LIN {X 0,Y 580.1,Z 304.268,A -85,B 0,C 180,E1 -1819.83,E2 -1819.83} C_VEL
LIN {X 0,Y 580.128,Z 300.119,A -85,B 0,C 180,E1 -1822.058,E2 -1822.058} C_VEL
LIN {X 0,Y 580.155,Z 294.555,A -85,B 0,C 180,E1 -1825.087,E2 -1825.087} C_VEL
LIN {X 0,Y 580.133,Z 290.01,A -85,B 0,C 180,E1 -1827.41,E2 -1827.41} C_VEL
LIN {X 0,Y 580.063,Z 285.03,A -85,B 0,C 180,E1 -1829.785,E2 -1829.785} C_VEL
LIN {X 0,Y 580.054,Z 279.379,A -85,B 0,C 180,E1 -1832.216,E2 -1832.216} C_VEL
LIN {X 0,Y 580.077,Z 277.233,A -85,B 0,C 180,E1 -1833.103,E2 -1833.103} C_VEL
LIN {X 0,Y 580.282,Z 277.204,A -85,B 0,C 180,E1 -1834.697,E2 -1834.697} C_VEL
LIN {X 0,Y 580.301,Z 277.201,A -85,B 0,C 180,E1 -1837.268,E2 -1837.268} C_VEL
LIN {X 0,Y 580.292,Z 277.205,A -85,B 0,C 180,E1 -1840.27,E2 -1840.27} C_VEL
LIN {X 0,Y 580.264,Z 277.206,A -85,B 0,C 180,E1 -1842.708,E2 -1842.708} C_VEL
LIN {X 0,Y 580.273,Z 277.208,A -85,B 0,C 180,E1 -1845.609,E2 -1845.609} C_VEL
LIN {X 0,Y 580.278,Z 277.204,A -85,B 0,C 180,E1 -1848.669,E2 -1848.669} C_VEL
LIN {X 0,Y 580.274,Z 277.208,A -85,B 0,C 180,E1 -1850.964,E2 -1850.964} C_VEL
LIN {X 0,Y 580.309,Z 277.247,A -85,B 0,C 180,E1 -1853.219,E2 -1853.219} C_VEL
LIN {X 0,Y 580.988,Z 281.668,A -85,B 0,C 180,E1 -1854.504,E2 -1854.504} C_VEL
LIN {X 0,Y 580.826,Z 290.876,A -85,B 0,C 180,E1 -1857.009,E2 -1857.009} C_VEL
LIN {X 0,Y 580.744,Z 300.085,A -85,B 0,C 180,E1 -1859.451,E2 -1859.451} C_VEL
LIN {X 0,Y 580.649,Z 311.291,A -85,B 0,C 180,E1 -1862.344,E2 -1862.344} C_VEL
LIN {X 0,Y 580.515,Z 321.571,A -85,B 0,C 180,E1 -1864.93,E2 -1864.93} C_VEL
LIN {X 0,Y 580.444,Z 332.314,A -85,B 0,C 180,E1 -1867.579,E2 -1867.579} C_VEL
LIN {X 0,Y 580.362,Z 343.058,A -85,B 0,C 180,E1 -1870.18,E2 -1870.18} C_VEL
LIN {X 0,Y 580.308,Z 355.336,A -85,B 0,C 180,E1 -1873.102,E2 -1873.102} C_VEL
LIN {X 0,Y 580.195,Z 367.614,A -85,B 0,C 180,E1 -1875.98,E2 -1875.98} C_VEL
LIN {X 0,Y 580.152,Z 374.712,A -85,B 0,C 180,E1 -1877.627,E2 -1877.627} C_VEL
LIN {X 0,Y 580.817,Z 380.085,A -85,B 0,C 180,E1 -1877.73,E2 -1877.73} C_VEL
LIN {X 0,Y 580.72,Z 393.734,A -85,B 0,C 180,E1 -1878.061,E2 -1878.061} C_VEL
LIN {X 0,Y 580.617,Z 406.32,A -85,B 0,C 180,E1 -1878.515,E2 -1878.515} C_VEL
LIN {X 0,Y 580.487,Z 418.208,A -85,B 0,C 180,E1 -1879.095,E2 -1879.095} C_VEL
LIN {X 0,Y 580.451,Z 429.476,A -85,B 0,C 180,E1 -1879.8,E2 -1879.8} C_VEL
LIN {X 0,Y 580.352,Z 439.646,A -85,B 0,C 180,E1 -1880.591,E2 -1880.591} C_VEL
LIN {X 0,Y 580.279,Z 448.787,A -85,B 0,C 180,E1 -1881.468,E2 -1881.468} C_VEL
LIN {X 0,Y 580.199,Z 457.691,A -85,B 0,C 180,E1 -1882.518,E2 -1882.518} C_VEL
LIN {X 0,Y 580.12,Z 464.465,A -85,B 0,C 180,E1 -1883.505,E2 -1883.505} C_VEL
LIN {X 0,Y 580.139,Z 469.68,A -85,B 0,C 180,E1 -1884.438,E2 -1884.438} C_VEL
LIN {X 0,Y 580.108,Z 474.371,A -85,B 0,C 180,E1 -1885.483,E2 -1885.483} C_VEL
LIN {X 0,Y 580.123,Z 477.956,A -85,B 0,C 180,E1 -1886.527,E2 -1886.527} C_VEL
LIN {X 0,Y 580.043,Z 479.809,A -85,B 0,C 180,E1 -1887.222,E2 -1887.222} C_VEL
LIN {X 0,Y 580.04,Z 481.201,A -85,B 0,C 180,E1 -1887.917,E2 -1887.917} C_VEL
LIN {X 0,Y 580.04,Z 482.784,A -85,B 0,C 180,E1 -1889.306,E2 -1889.306} C_VEL
LIN {X 0,Y 580.037,Z 483,A -85,B 0,C 180,E1 -1890,E2 -1890} C_VEL
LIN {X 0,Y 580.047,Z 482.185,A -85,B 0,C 180,E1 -1891.389,E2 -1891.389} C_VEL
LIN {X 0,Y 580.04,Z 481.202,A -85,B 0,C 180,E1 -1892.083,E2 -1892.083} C_VEL
LIN {X 0,Y 580.043,Z 479.809,A -85,B 0,C 180,E1 -1892.778,E2 -1892.778} C_VEL
LIN {X 0,Y 580.11,Z 476.896,A -85,B 0,C 180,E1 -1893.821,E2 -1893.821} C_VEL
LIN {X 0,Y 580.053,Z 472.949,A -85,B 0,C 180,E1 -1894.865,E2 -1894.865} C_VEL
LIN {X 0,Y 580.139,Z 466.877,A -85,B 0,C 180,E1 -1896.085,E2 -1896.085} C_VEL
LIN {X 0,Y 580.184,Z 460.236,A -85,B 0,C 180,E1 -1897.132,E2 -1897.132} C_VEL
LIN {X 0,Y 580.25,Z 451.989,A -85,B 0,C 180,E1 -1898.182,E2 -1898.182} C_VEL
LIN {X 0,Y 580.308,Z 443.537,A -85,B 0,C 180,E1 -1899.058,E2 -1899.058} C_VEL
LIN {X 0,Y 580.417,Z 433.093,A -85,B 0,C 180,E1 -1899.936,E2 -1899.936} C_VEL
LIN {X 0,Y 580.475,Z 422.758,A -85,B 0,C 180,E1 -1900.64,E2 -1900.64} C_VEL
LIN {X 0,Y 580.563,Z 411.592,A -85,B 0,C 180,E1 -1901.248,E2 -1901.248} C_VEL
LIN {X 0,Y 580.628,Z 399.765,A -85,B 0,C 180,E1 -1901.742,E2 -1901.742} C_VEL
LIN {X 0,Y 580.766,Z 386.349,A -85,B 0,C 180,E1 -1902.138,E2 -1902.138} C_VEL
LIN {X 0,Y 580.611,Z 377.609,A -85,B 0,C 180,E1 -1902.318,E2 -1902.318} C_VEL
LIN {X 0,Y 580.153,Z 374.712,A -85,B 0,C 180,E1 -1902.373,E2 -1902.373} C_VEL
LIN {X 0,Y 580.234,Z 363.009,A -85,B 0,C 180,E1 -1905.095,E2 -1905.095} C_VEL
LIN {X 0,Y 580.326,Z 350.731,A -85,B 0,C 180,E1 -1907.988,E2 -1907.988} C_VEL
LIN {X 0,Y 580.403,Z 338.679,A -85,B 0,C 180,E1 -1910.874,E2 -1910.874} C_VEL
LIN {X 0,Y 580.49,Z 327.71,A -85,B 0,C 180,E1 -1913.549,E2 -1913.549} C_VEL
LIN {X 0,Y 580.586,Z 315.432,A -85,B 0,C 180,E1 -1916.608,E2 -1916.608} C_VEL
LIN {X 0,Y 580.721,Z 304.562,A -85,B 0,C 180,E1 -1919.383,E2 -1919.383} C_VEL
LIN {X 0,Y 580.825,Z 293.946,A -85,B 0,C 180,E1 -1922.168,E2 -1922.168} C_VEL
LIN {X 0,Y 580.893,Z 284.737,A -85,B 0,C 180,E1 -1924.655,E2 -1924.655} C_VEL
LIN {X 0,Y 580.881,Z 280.446,A -85,B 0,C 180,E1 -1925.843,E2 -1925.843} C_VEL
LIN {X 0,Y 580.27,Z 277.208,A -85,B 0,C 180,E1 -1926.827,E2 -1926.827} C_VEL
LIN {X 0,Y 580.284,Z 277.205,A -85,B 0,C 180,E1 -1929.184,E2 -1929.184} C_VEL
LIN {X 0,Y 580.252,Z 277.203,A -85,B 0,C 180,E1 -1931.771,E2 -1931.771} C_VEL
LIN {X 0,Y 580.248,Z 277.211,A -85,B 0,C 180,E1 -1934.628,E2 -1934.628} C_VEL
LIN {X 0,Y 580.263,Z 277.201,A -85,B 0,C 180,E1 -1937.292,E2 -1937.292} C_VEL
LIN {X 0,Y 580.297,Z 277.203,A -85,B 0,C 180,E1 -1940.067,E2 -1940.067} C_VEL
LIN {X 0,Y 580.301,Z 277.196,A -85,B 0,C 180,E1 -1943.066,E2 -1943.066} C_VEL
LIN {X 0,Y 580.317,Z 277.2,A -85,B 0,C 180,E1 -1946.145,E2 -1946.145} C_VEL
LIN {X 0,Y 580.278,Z 277.199,A -85,B 0,C 180,E1 -1948.615,E2 -1948.615} C_VEL
LIN {X 0,Y 580.296,Z 277.199,A -85,B 0,C 180,E1 -1951.024,E2 -1951.024} C_VEL
LIN {X 0,Y 580.293,Z 277.204,A -85,B 0,C 180,E1 -1953.666,E2 -1953.666} C_VEL
LIN {X 0,Y 580.149,Z 277.224,A -85,B 0,C 180,E1 -1956.436,E2 -1956.436} C_VEL
LIN {X 0,Y 580.074,Z 277.231,A -85,B 0,C 180,E1 -1957.188,E2 -1957.188} C_VEL
LIN {X 0,Y 580.081,Z 279.813,A -85,B 0,C 180,E1 -1959.43,E2 -1959.43} C_VEL
LIN {X 0,Y 580.033,Z 283.328,A -85,B 0,C 180,E1 -1962.367,E2 -1962.367} C_VEL
LIN {X 0,Y 580.047,Z 285.965,A -85,B 0,C 180,E1 -1964.54,E2 -1964.54} C_VEL
LIN {X 0,Y 580.045,Z 288.602,A -85,B 0,C 180,E1 -1966.691,E2 -1966.691} C_VEL
LIN {X 0,Y 580.043,Z 290.118,A -85,B 0,C 180,E1 -1967.758,E2 -1967.758} C_VEL
LIN {X 0,Y 580.785,Z 296.369,A -85,B 0,C 180,E1 -1967.907,E2 -1967.907} C_VEL
LIN {X 0,Y 580.646,Z 309.747,A -85,B 0,C 180,E1 -1968.303,E2 -1968.303} C_VEL
LIN {X 0,Y 580.564,Z 320.592,A -85,B 0,C 180,E1 -1968.752,E2 -1968.752} C_VEL
LIN {X 0,Y 580.493,Z 331.974,A -85,B 0,C 180,E1 -1969.36,E2 -1969.36} C_VEL
LIN {X 0,Y 580.42,Z 342.507,A -85,B 0,C 180,E1 -1970.064,E2 -1970.064} C_VEL
LIN {X 0,Y 580.319,Z 353.054,A -85,B 0,C 180,E1 -1970.942,E2 -1970.942} C_VEL
LIN {X 0,Y 580.251,Z 361.571,A -85,B 0,C 180,E1 -1971.818,E2 -1971.818} C_VEL
LIN {X 0,Y 580.176,Z 368.64,A -85,B 0,C 180,E1 -1972.693,E2 -1972.693} C_VEL
LIN {X 0,Y 580.137,Z 375.587,A -85,B 0,C 180,E1 -1973.741,E2 -1973.741} C_VEL
LIN {X 0,Y 580.086,Z 381.161,A -85,B 0,C 180,E1 -1974.787,E2 -1974.787} C_VEL
LIN {X 0,Y 580.105,Z 385.527,A -85,B 0,C 180,E1 -1975.831,E2 -1975.831} C_VEL
LIN {X 0,Y 580.043,Z 389.694,A -85,B 0,C 180,E1 -1977.222,E2 -1977.222} C_VEL
LIN {X 0,Y 580.04,Z 391.135,A -85,B 0,C 180,E1 -1977.917,E2 -1977.917} C_VEL
LIN {X 0,Y 580.04,Z 392.757,A -85,B 0,C 180,E1 -1979.306,E2 -1979.306} C_VEL
LIN {X 0,Y 580.038,Z 392.996,A -85,B 0,C 180,E1 -1980,E2 -1980} C_VEL
LIN {X 0,Y 580.047,Z 392.229,A -85,B 0,C 180,E1 -1981.389,E2 -1981.389} C_VEL
LIN {X 0,Y 580.04,Z 391.278,A -85,B 0,C 180,E1 -1982.083,E2 -1982.083} C_VEL
LIN {X 0,Y 580.044,Z 389.883,A -85,B 0,C 180,E1 -1982.778,E2 -1982.778} C_VEL
LIN {X 0,Y 580.11,Z 387.011,A -85,B 0,C 180,E1 -1983.821,E2 -1983.821} C_VEL
LIN {X 0,Y 580.053,Z 383.122,A -85,B 0,C 180,E1 -1984.865,E2 -1984.865} C_VEL
LIN {X 0,Y 580.161,Z 378.1,A -85,B 0,C 180,E1 -1985.91,E2 -1985.91} C_VEL
LIN {X 0,Y 580.158,Z 371.776,A -85,B 0,C 180,E1 -1986.958,E2 -1986.958} C_VEL
LIN {X 0,Y 580.231,Z 363.836,A -85,B 0,C 180,E1 -1988.007,E2 -1988.007} C_VEL
LIN {X 0,Y 580.298,Z 355.752,A -85,B 0,C 180,E1 -1988.883,E2 -1988.883} C_VEL
LIN {X 0,Y 580.366,Z 345.921,A -85,B 0,C 180,E1 -1989.761,E2 -1989.761} C_VEL
LIN {X 0,Y 580.459,Z 334.898,A -85,B 0,C 180,E1 -1990.552,E2 -1990.552} C_VEL
LIN {X 0,Y 580.522,Z 324.063,A -85,B 0,C 180,E1 -1991.169,E2 -1991.169} C_VEL
LIN {X 0,Y 580.626,Z 312.523,A -85,B 0,C 180,E1 -1991.68,E2 -1991.68} C_VEL
LIN {X 0,Y 580.725,Z 300.605,A -85,B 0,C 180,E1 -1992.072,E2 -1992.072} C_VEL
LIN {X 0,Y 580.652,Z 293.717,A -85,B 0,C 180,E1 -1992.245,E2 -1992.245} C_VEL
LIN {X 0,Y 580.063,Z 289.894,A -85,B 0,C 180,E1 -1992.352,E2 -1992.352} C_VEL
LIN {X 0,Y 580.004,Z 286.954,A -85,B 0,C 180,E1 -1994.742,E2 -1994.742} C_VEL
LIN {X 0,Y 580.022,Z 283.684,A -85,B 0,C 180,E1 -1997.429,E2 -1997.429} C_VEL
LIN {X 0,Y 579.37,Z 283.014,A -85,B 0,C 180,E1 -1998.005,E2 -1998.005} C_VEL
LIN {X 0,Y 576.505,Z 282.007,A -85,B 0,C 180,E1 -1998.941,E2 -1998.941} C_VEL
LIN {X 0,Y 574.078,Z 281.214,A -85,B 0,C 180,E1 -1999.694,E2 -1999.694} C_VEL
LIN {X 0,Y 573.042,Z 280.574,A -85,B 0,C 180,E1 -2000.275,E2 -2000.275} C_VEL
LIN {X 0,Y 572.962,Z 280.347,A -85,B 0,C 180,E1 -2000.472,E2 -2000.472} C_VEL
LIN {X 0,Y 572.945,Z 278.247,A -85,B 0,C 180,E1 -2002.35,E2 -2002.35} C_VEL
LIN {X 0,Y 573.197,Z 278.087,A -85,B 0,C 180,E1 -2004.862,E2 -2004.862} C_VEL
LIN {X 0,Y 573.223,Z 278.081,A -85,B 0,C 180,E1 -2006.978,E2 -2006.978} C_VEL
LIN {X 0,Y 573.244,Z 278.074,A -85,B 0,C 180,E1 -2009.487,E2 -2009.487} C_VEL
LIN {X 0,Y 573.257,Z 278.078,A -85,B 0,C 180,E1 -2012.645,E2 -2012.645} C_VEL
LIN {X 0,Y 573.208,Z 278.078,A -85,B 0,C 180,E1 -2015.188,E2 -2015.188} C_VEL
LIN {X 0,Y 573.24,Z 278.079,A -85,B 0,C 180,E1 -2017.807,E2 -2017.807} C_VEL
LIN {X 0,Y 573.248,Z 278.077,A -85,B 0,C 180,E1 -2020.525,E2 -2020.525} C_VEL
LIN {X 0,Y 573.243,Z 278.076,A -85,B 0,C 180,E1 -2023.359,E2 -2023.359} C_VEL
LIN {X 0,Y 573.248,Z 278.076,A -85,B 0,C 180,E1 -2026.331,E2 -2026.331} C_VEL
LIN {X 0,Y 573.238,Z 278.076,A -85,B 0,C 180,E1 -2028.543,E2 -2028.543} C_VEL
LIN {X 0,Y 573.245,Z 278.078,A -85,B 0,C 180,E1 -2031.298,E2 -2031.298} C_VEL
LIN {X 0,Y 573.216,Z 278.082,A -85,B 0,C 180,E1 -2034.019,E2 -2034.019} C_VEL
LIN {X 0,Y 573.166,Z 278.255,A -85,B 0,C 180,E1 -2035.771,E2 -2035.771} C_VEL
LIN {X 0,Y 573.104,Z 282.816,A -85,B 0,C 180,E1 -2038.176,E2 -2038.176} C_VEL
LIN {X 0,Y 573.057,Z 287.256,A -85,B 0,C 180,E1 -2040.622,E2 -2040.622} C_VEL
LIN {X 0,Y 573.058,Z 291.597,A -85,B 0,C 180,E1 -2043.014,E2 -2043.014} C_VEL
LIN {X 0,Y 573.07,Z 295.867,A -85,B 0,C 180,E1 -2045.357,E2 -2045.357} C_VEL
LIN {X 0,Y 573.042,Z 299.961,A -85,B 0,C 180,E1 -2047.654,E2 -2047.654} C_VEL
LIN {X 0,Y 573.016,Z 304.101,A -85,B 0,C 180,E1 -2049.915,E2 -2049.915} C_VEL
LIN {X 0,Y 572.975,Z 308.248,A -85,B 0,C 180,E1 -2052.143,E2 -2052.143} C_VEL
LIN {X 0,Y 573,Z 313.778,A -85,B 0,C 180,E1 -2055.074,E2 -2055.074} C_VEL
LIN {X 0,Y 573.003,Z 318.682,A -85,B 0,C 180,E1 -2057.583,E2 -2057.583} C_VEL
LIN {X 0,Y 573.854,Z 325.38,A -85,B 0,C 180,E1 -2057.736,E2 -2057.736} C_VEL
LIN {X 0,Y 573.74,Z 337.077,A -85,B 0,C 180,E1 -2058.07,E2 -2058.07} C_VEL
LIN {X 0,Y 573.601,Z 347.726,A -85,B 0,C 180,E1 -2058.484,E2 -2058.484} C_VEL
LIN {X 0,Y 573.525,Z 359.272,A -85,B 0,C 180,E1 -2059.068,E2 -2059.068} C_VEL
LIN {X 0,Y 573.444,Z 371.328,A -85,B 0,C 180,E1 -2059.853,E2 -2059.853} C_VEL
LIN {X 0,Y 573.321,Z 381.079,A -85,B 0,C 180,E1 -2060.652,E2 -2060.652} C_VEL
LIN {X 0,Y 573.225,Z 389.959,A -85,B 0,C 180,E1 -2061.54,E2 -2061.54} C_VEL
LIN {X 0,Y 573.143,Z 397.316,A -85,B 0,C 180,E1 -2062.425,E2 -2062.425} C_VEL
LIN {X 0,Y 573.104,Z 403.818,A -85,B 0,C 180,E1 -2063.369,E2 -2063.369} C_VEL
LIN {X 0,Y 573.07,Z 409.452,A -85,B 0,C 180,E1 -2064.37,E2 -2064.37} C_VEL
LIN {X 0,Y 573.028,Z 414.2,A -85,B 0,C 180,E1 -2065.427,E2 -2065.427} C_VEL
LIN {X 0,Y 573.022,Z 417.834,A -85,B 0,C 180,E1 -2066.484,E2 -2066.484} C_VEL
LIN {X 0,Y 572.959,Z 419.672,A -85,B 0,C 180,E1 -2067.188,E2 -2067.188} C_VEL
LIN {X 0,Y 572.946,Z 422.142,A -85,B 0,C 180,E1 -2068.594,E2 -2068.594} C_VEL
LIN {X 0,Y 572.941,Z 422.751,A -85,B 0,C 180,E1 -2069.297,E2 -2069.297} C_VEL
LIN {X 0,Y 572.94,Z 422.811,A -85,B 0,C 180,E1 -2070.703,E2 -2070.703} C_VEL
LIN {X 0,Y 572.947,Z 422.242,A -85,B 0,C 180,E1 -2071.406,E2 -2071.406} C_VEL
LIN {X 0,Y 572.96,Z 419.898,A -85,B 0,C 180,E1 -2072.812,E2 -2072.812} C_VEL
LIN {X 0,Y 573.015,Z 417.024,A -85,B 0,C 180,E1 -2073.868,E2 -2073.868} C_VEL
LIN {X 0,Y 572.962,Z 413.114,A -85,B 0,C 180,E1 -2074.926,E2 -2074.926} C_VEL
LIN {X 0,Y 573.076,Z 408.064,A -85,B 0,C 180,E1 -2075.983,E2 -2075.983} C_VEL
LIN {X 0,Y 573.082,Z 401.729,A -85,B 0,C 180,E1 -2077.044,E2 -2077.044} C_VEL
LIN {X 0,Y 573.175,Z 393.872,A -85,B 0,C 180,E1 -2078.106,E2 -2078.106} C_VEL
LIN {X 0,Y 573.287,Z 383.962,A -85,B 0,C 180,E1 -2079.17,E2 -2079.17} C_VEL
LIN {X 0,Y 573.395,Z 374.773,A -85,B 0,C 180,E1 -2079.97,E2 -2079.97} C_VEL
LIN {X 0,Y 573.466,Z 364.905,A -85,B 0,C 180,E1 -2080.678,E2 -2080.678} C_VEL
LIN {X 0,Y 573.561,Z 352.657,A -85,B 0,C 180,E1 -2081.379,E2 -2081.379} C_VEL
LIN {X 0,Y 573.709,Z 339.914,A -85,B 0,C 180,E1 -2081.921,E2 -2081.921} C_VEL
LIN {X 0,Y 573.809,Z 328.042,A -85,B 0,C 180,E1 -2082.287,E2 -2082.287} C_VEL
LIN {X 0,Y 573.654,Z 322.803,A -85,B 0,C 180,E1 -2082.418,E2 -2082.418} C_VEL
LIN {X 0,Y 572.975,Z 318.53,A -85,B 0,C 180,E1 -2082.53,E2 -2082.53} C_VEL
LIN {X 0,Y 572.999,Z 313.949,A -85,B 0,C 180,E1 -2084.926,E2 -2084.926} C_VEL
LIN {X 0,Y 572.97,Z 308.416,A -85,B 0,C 180,E1 -2087.857,E2 -2087.857} C_VEL
LIN {X 0,Y 573.017,Z 304.267,A -85,B 0,C 180,E1 -2090.085,E2 -2090.085} C_VEL
LIN {X 0,Y 573.043,Z 300.122,A -85,B 0,C 180,E1 -2092.346,E2 -2092.346} C_VEL
LIN {X 0,Y 573.087,Z 294.611,A -85,B 0,C 180,E1 -2095.418,E2 -2095.418} C_VEL
LIN {X 0,Y 573.082,Z 289.95,A -85,B 0,C 180,E1 -2097.996,E2 -2097.996} C_VEL
LIN {X 0,Y 573.111,Z 284.493,A -85,B 0,C 180,E1 -2101,E2 -2101} C_VEL
LIN {X 0,Y 573.14,Z 279.854,A -85,B 0,C 180,E1 -2103.505,E2 -2103.505} C_VEL
LIN {X 0,Y 573.186,Z 278.091,A -85,B 0,C 180,E1 -2104.494,E2 -2104.494} C_VEL
LIN {X 0,Y 573.241,Z 278.084,A -85,B 0,C 180,E1 -2107.164,E2 -2107.164} C_VEL
LIN {X 0,Y 573.25,Z 278.081,A -85,B 0,C 180,E1 -2109.607,E2 -2109.607} C_VEL
LIN {X 0,Y 573.245,Z 278.081,A -85,B 0,C 180,E1 -2112.642,E2 -2112.642} C_VEL
LIN {X 0,Y 573.226,Z 278.082,A -85,B 0,C 180,E1 -2115.665,E2 -2115.665} C_VEL
LIN {X 0,Y 573.229,Z 278.082,A -85,B 0,C 180,E1 -2118.543,E2 -2118.543} C_VEL
LIN {X 0,Y 573.248,Z 278.081,A -85,B 0,C 180,E1 -2121.299,E2 -2121.299} C_VEL
LIN {X 0,Y 573.197,Z 278.089,A -85,B 0,C 180,E1 -2124.021,E2 -2124.021} C_VEL
LIN {X 0,Y 573.16,Z 278.132,A -85,B 0,C 180,E1 -2125.781,E2 -2125.781} C_VEL
LIN {X 0,Y 573.11,Z 284.453,A -85,B 0,C 180,E1 -2129.138,E2 -2129.138} C_VEL
LIN {X 0,Y 573.098,Z 290.134,A -85,B 0,C 180,E1 -2132.225,E2 -2132.225} C_VEL
LIN {X 0,Y 573.099,Z 295.565,A -85,B 0,C 180,E1 -2135.159,E2 -2135.159} C_VEL
LIN {X 0,Y 573.042,Z 299.964,A -85,B 0,C 180,E1 -2137.654,E2 -2137.654} C_VEL
LIN {X 0,Y 573.016,Z 304.101,A -85,B 0,C 180,E1 -2139.915,E2 -2139.915} C_VEL
LIN {X 0,Y 572.975,Z 308.248,A -85,B 0,C 180,E1 -2142.143,E2 -2142.143} C_VEL
LIN {X 0,Y 573,Z 313.777,A -85,B 0,C 180,E1 -2145.074,E2 -2145.074} C_VEL
LIN {X 0,Y 573.003,Z 318.741,A -85,B 0,C 180,E1 -2147.583,E2 -2147.583} C_VEL
LIN {X 0,Y 573.856,Z 325.326,A -85,B 0,C 180,E1 -2147.736,E2 -2147.736} C_VEL
LIN {X 0,Y 573.733,Z 337.39,A -85,B 0,C 180,E1 -2148.079,E2 -2148.079} C_VEL
LIN {X 0,Y 573.626,Z 349.625,A -85,B 0,C 180,E1 -2148.566,E2 -2148.566} C_VEL
LIN {X 0,Y 573.533,Z 360.687,A -85,B 0,C 180,E1 -2149.149,E2 -2149.149} C_VEL
LIN {X 0,Y 573.419,Z 371.271,A -85,B 0,C 180,E1 -2149.852,E2 -2149.852} C_VEL
LIN {X 0,Y 573.312,Z 379.078,A -85,B 0,C 180,E1 -2150.474,E2 -2150.474} C_VEL
LIN {X 0,Y 573.216,Z 388.327,A -85,B 0,C 180,E1 -2151.362,E2 -2151.362} C_VEL
LIN {X 0,Y 573.161,Z 395.962,A -85,B 0,C 180,E1 -2152.248,E2 -2152.248} C_VEL
LIN {X 0,Y 573.09,Z 403.915,A -85,B 0,C 180,E1 -2153.381,E2 -2153.381} C_VEL
LIN {X 0,Y 573.071,Z 409.462,A -85,B 0,C 180,E1 -2154.37,E2 -2154.37} C_VEL
LIN {X 0,Y 573.028,Z 414.203,A -85,B 0,C 180,E1 -2155.427,E2 -2155.427} C_VEL
LIN {X 0,Y 573.022,Z 417.833,A -85,B 0,C 180,E1 -2156.484,E2 -2156.484} C_VEL
LIN {X 0,Y 572.959,Z 419.688,A -85,B 0,C 180,E1 -2157.188,E2 -2157.188} C_VEL
LIN {X 0,Y 572.946,Z 422.135,A -85,B 0,C 180,E1 -2158.594,E2 -2158.594} C_VEL
LIN {X 0,Y 572.941,Z 422.758,A -85,B 0,C 180,E1 -2159.297,E2 -2159.297} C_VEL
LIN {X 0,Y 572.94,Z 422.805,A -85,B 0,C 180,E1 -2160.703,E2 -2160.703} C_VEL
LIN {X 0,Y 572.947,Z 422.244,A -85,B 0,C 180,E1 -2161.406,E2 -2161.406} C_VEL
LIN {X 0,Y 572.96,Z 419.895,A -85,B 0,C 180,E1 -2162.812,E2 -2162.812} C_VEL
LIN {X 0,Y 573.015,Z 417.023,A -85,B 0,C 180,E1 -2163.868,E2 -2163.868} C_VEL
LIN {X 0,Y 572.962,Z 413.115,A -85,B 0,C 180,E1 -2164.926,E2 -2164.926} C_VEL
LIN {X 0,Y 573.076,Z 408.065,A -85,B 0,C 180,E1 -2165.983,E2 -2165.983} C_VEL
LIN {X 0,Y 573.082,Z 401.724,A -85,B 0,C 180,E1 -2167.044,E2 -2167.044} C_VEL
LIN {X 0,Y 573.175,Z 393.869,A -85,B 0,C 180,E1 -2168.106,E2 -2168.106} C_VEL
LIN {X 0,Y 573.282,Z 383.983,A -85,B 0,C 180,E1 -2169.17,E2 -2169.17} C_VEL
LIN {X 0,Y 573.395,Z 374.778,A -85,B 0,C 180,E1 -2169.97,E2 -2169.97} C_VEL
LIN {X 0,Y 573.465,Z 364.906,A -85,B 0,C 180,E1 -2170.676,E2 -2170.676} C_VEL
LIN {X 0,Y 573.551,Z 354.024,A -85,B 0,C 180,E1 -2171.306,E2 -2171.306} C_VEL
LIN {X 0,Y 573.678,Z 341.003,A -85,B 0,C 180,E1 -2171.886,E2 -2171.886} C_VEL
LIN {X 0,Y 573.809,Z 328.053,A -85,B 0,C 180,E1 -2172.287,E2 -2172.287} C_VEL
LIN {X 0,Y 573.654,Z 322.819,A -85,B 0,C 180,E1 -2172.418,E2 -2172.418} C_VEL
LIN {X 0,Y 572.975,Z 318.53,A -85,B 0,C 180,E1 -2172.53,E2 -2172.53} C_VEL
LIN {X 0,Y 572.999,Z 313.949,A -85,B 0,C 180,E1 -2174.926,E2 -2174.926} C_VEL
LIN {X 0,Y 572.97,Z 308.416,A -85,B 0,C 180,E1 -2177.857,E2 -2177.857} C_VEL
LIN {X 0,Y 573.017,Z 304.267,A -85,B 0,C 180,E1 -2180.085,E2 -2180.085} C_VEL
LIN {X 0,Y 573.044,Z 300.135,A -85,B 0,C 180,E1 -2182.346,E2 -2182.346} C_VEL
LIN {X 0,Y 573.072,Z 295.562,A -85,B 0,C 180,E1 -2184.835,E2 -2184.835} C_VEL
LIN {X 0,Y 573.053,Z 291.375,A -85,B 0,C 180,E1 -2186.986,E2 -2186.986} C_VEL
LIN {X 0,Y 572.981,Z 286.225,A -85,B 0,C 180,E1 -2189.441,E2 -2189.441} C_VEL
LIN {X 0,Y 572.987,Z 280.726,A -85,B 0,C 180,E1 -2191.831,E2 -2191.831} C_VEL
LIN {X 0,Y 572.991,Z 278.115,A -85,B 0,C 180,E1 -2192.923,E2 -2192.923} C_VEL
LIN {X 0,Y 573.228,Z 278.083,A -85,B 0,C 180,E1 -2194.77,E2 -2194.77} C_VEL
LIN {X 0,Y 573.236,Z 278.084,A -85,B 0,C 180,E1 -2197.808,E2 -2197.808} C_VEL
LIN {X 0,Y 573.248,Z 278.082,A -85,B 0,C 180,E1 -2200.525,E2 -2200.525} C_VEL
LIN {X 0,Y 573.244,Z 278.08,A -85,B 0,C 180,E1 -2203.669,E2 -2203.669} C_VEL
LIN {X 0,Y 573.235,Z 278.081,A -85,B 0,C 180,E1 -2206.64,E2 -2206.64} C_VEL
LIN {X 0,Y 573.247,Z 278.083,A -85,B 0,C 180,E1 -2209.475,E2 -2209.475} C_VEL
LIN {X 0,Y 573.236,Z 278.084,A -85,B 0,C 180,E1 -2212.192,E2 -2212.192} C_VEL
LIN {X 0,Y 573.263,Z 278.145,A -85,B 0,C 180,E1 -2212.957,E2 -2212.957} C_VEL
LIN {X 0,Y 574.098,Z 283.202,A -85,B 0,C 180,E1 -2214.445,E2 -2214.445} C_VEL
LIN {X 0,Y 573.899,Z 292.411,A -85,B 0,C 180,E1 -2216.979,E2 -2216.979} C_VEL
LIN {X 0,Y 573.794,Z 301.619,A -85,B 0,C 180,E1 -2219.449,E2 -2219.449} C_VEL
LIN {X 0,Y 573.677,Z 312.363,A -85,B 0,C 180,E1 -2222.255,E2 -2222.255} C_VEL
LIN {X 0,Y 573.517,Z 323.417,A -85,B 0,C 180,E1 -2225.069,E2 -2225.069} C_VEL
LIN {X 0,Y 573.42,Z 333.849,A -85,B 0,C 180,E1 -2227.67,E2 -2227.67} C_VEL
LIN {X 0,Y 573.329,Z 346.127,A -85,B 0,C 180,E1 -2230.672,E2 -2230.672} C_VEL
LIN {X 0,Y 573.257,Z 357.095,A -85,B 0,C 180,E1 -2233.309,E2 -2233.309} C_VEL
LIN {X 0,Y 573.153,Z 369.148,A -85,B 0,C 180,E1 -2236.166,E2 -2236.166} C_VEL
LIN {X 0,Y 573.108,Z 374.712,A -85,B 0,C 180,E1 -2237.473,E2 -2237.473} C_VEL
LIN {X 0,Y 573.891,Z 381.227,A -85,B 0,C 180,E1 -2237.603,E2 -2237.603} C_VEL
LIN {X 0,Y 573.775,Z 394.495,A -85,B 0,C 180,E1 -2237.937,E2 -2237.937} C_VEL
LIN {X 0,Y 573.644,Z 407.393,A -85,B 0,C 180,E1 -2238.421,E2 -2238.421} C_VEL
LIN {X 0,Y 573.52,Z 419.994,A -85,B 0,C 180,E1 -2239.063,E2 -2239.063} C_VEL
LIN {X 0,Y 573.45,Z 430.746,A -85,B 0,C 180,E1 -2239.764,E2 -2239.764} C_VEL
LIN {X 0,Y 573.308,Z 439.646,A -85,B 0,C 180,E1 -2240.474,E2 -2240.474} C_VEL
LIN {X 0,Y 573.215,Z 448.787,A -85,B 0,C 180,E1 -2241.362,E2 -2241.362} C_VEL
LIN {X 0,Y 573.142,Z 457.69,A -85,B 0,C 180,E1 -2242.425,E2 -2242.425} C_VEL
LIN {X 0,Y 573.051,Z 464.405,A -85,B 0,C 180,E1 -2243.415,E2 -2243.415} C_VEL
LIN {X 0,Y 573.07,Z 469.68,A -85,B 0,C 180,E1 -2244.37,E2 -2244.37} C_VEL
LIN {X 0,Y 573.028,Z 474.371,A -85,B 0,C 180,E1 -2245.427,E2 -2245.427} C_VEL
LIN {X 0,Y 573.022,Z 477.956,A -85,B 0,C 180,E1 -2246.484,E2 -2246.484} C_VEL
LIN {X 0,Y 572.959,Z 479.809,A -85,B 0,C 180,E1 -2247.188,E2 -2247.188} C_VEL
LIN {X 0,Y 572.94,Z 481.201,A -85,B 0,C 180,E1 -2247.891,E2 -2247.891} C_VEL
LIN {X 0,Y 572.941,Z 482.784,A -85,B 0,C 180,E1 -2249.297,E2 -2249.297} C_VEL
LIN {X 0,Y 572.938,Z 483,A -85,B 0,C 180,E1 -2250,E2 -2250} C_VEL
LIN {X 0,Y 572.946,Z 482.185,A -85,B 0,C 180,E1 -2251.406,E2 -2251.406} C_VEL
LIN {X 0,Y 572.94,Z 481.201,A -85,B 0,C 180,E1 -2252.109,E2 -2252.109} C_VEL
LIN {X 0,Y 572.959,Z 479.81,A -85,B 0,C 180,E1 -2252.812,E2 -2252.812} C_VEL
LIN {X 0,Y 573.015,Z 476.896,A -85,B 0,C 180,E1 -2253.868,E2 -2253.868} C_VEL
LIN {X 0,Y 572.963,Z 472.949,A -85,B 0,C 180,E1 -2254.926,E2 -2254.926} C_VEL
LIN {X 0,Y 573.065,Z 466.877,A -85,B 0,C 180,E1 -2256.16,E2 -2256.16} C_VEL
LIN {X 0,Y 573.119,Z 460.236,A -85,B 0,C 180,E1 -2257.221,E2 -2257.221} C_VEL
LIN {X 0,Y 573.201,Z 451.989,A -85,B 0,C 180,E1 -2258.283,E2 -2258.283} C_VEL
LIN {X 0,Y 573.287,Z 443.537,A -85,B 0,C 180,E1 -2259.17,E2 -2259.17} C_VEL
LIN {X 0,Y 573.425,Z 433.093,A -85,B 0,C 180,E1 -2260.058,E2 -2260.058} C_VEL
LIN {X 0,Y 573.511,Z 421.536,A -85,B 0,C 180,E1 -2260.847,E2 -2260.847} C_VEL
LIN {X 0,Y 573.611,Z 409.878,A -85,B 0,C 180,E1 -2261.466,E2 -2261.466} C_VEL
LIN {X 0,Y 573.75,Z 397.174,A -85,B 0,C 180,E1 -2261.974,E2 -2261.974} C_VEL
LIN {X 0,Y 573.846,Z 384.519,A -85,B 0,C 180,E1 -2262.331,E2 -2262.331} C_VEL
LIN {X 0,Y 573.661,Z 378.329,A -85,B 0,C 180,E1 -2262.459,E2 -2262.459} C_VEL
LIN {X 0,Y 573.108,Z 374.712,A -85,B 0,C 180,E1 -2262.527,E2 -2262.527} C_VEL
LIN {X 0,Y 573.191,Z 363.009,A -85,B 0,C 180,E1 -2265.285,E2 -2265.285} C_VEL
LIN {X 0,Y 573.286,Z 352.266,A -85,B 0,C 180,E1 -2267.847,E2 -2267.847} C_VEL
LIN {X 0,Y 573.367,Z 339.988,A -85,B 0,C 180,E1 -2270.822,E2 -2270.822} C_VEL
LIN {X 0,Y 573.502,Z 327.71,A -85,B 0,C 180,E1 -2273.854,E2 -2273.854} C_VEL
LIN {X 0,Y 573.598,Z 316.972,A -85,B 0,C 180,E1 -2276.564,E2 -2276.564} C_VEL
LIN {X 0,Y 573.746,Z 306.224,A -85,B 0,C 180,E1 -2279.339,E2 -2279.339} C_VEL
LIN {X 0,Y 573.902,Z 294.954,A -85,B 0,C 180,E1 -2282.331,E2 -2282.331} C_VEL
LIN {X 0,Y 574.02,Z 285.623,A -85,B 0,C 180,E1 -2284.884,E2 -2284.884} C_VEL
LIN {X 0,Y 573.857,Z 281.439,A -85,B 0,C 180,E1 -2286.07,E2 -2286.07} C_VEL
LIN {X 0,Y 573.259,Z 278.082,A -85,B 0,C 180,E1 -2287.103,E2 -2287.103} C_VEL
LIN {X 0,Y 573.231,Z 278.079,A -85,B 0,C 180,E1 -2289.609,E2 -2289.609} C_VEL
LIN {X 0,Y 573.221,Z 278.086,A -85,B 0,C 180,E1 -2292.639,E2 -2292.639} C_VEL
LIN {X 0,Y 573.225,Z 278.078,A -85,B 0,C 180,E1 -2295.665,E2 -2295.665} C_VEL
LIN {X 0,Y 573.227,Z 278.084,A -85,B 0,C 180,E1 -2298.543,E2 -2298.543} C_VEL
LIN {X 0,Y 573.248,Z 278.075,A -85,B 0,C 180,E1 -2301.299,E2 -2301.299} C_VEL
LIN {X 0,Y 573.215,Z 278.087,A -85,B 0,C 180,E1 -2304.019,E2 -2304.019} C_VEL
LIN {X 0,Y 573.273,Z 278.073,A -85,B 0,C 180,E1 -2306.518,E2 -2306.518} C_VEL
LIN {X 0,Y 573.231,Z 278.079,A -85,B 0,C 180,E1 -2309.118,E2 -2309.118} C_VEL
LIN {X 0,Y 573.242,Z 278.083,A -85,B 0,C 180,E1 -2311.436,E2 -2311.436} C_VEL
LIN {X 0,Y 573.265,Z 278.078,A -85,B 0,C 180,E1 -2313.81,E2 -2313.81} C_VEL
LIN {X 0,Y 573.129,Z 278.097,A -85,B 0,C 180,E1 -2316.13,E2 -2316.13} C_VEL
LIN {X 0,Y 572.969,Z 278.362,A -85,B 0,C 180,E1 -2317.651,E2 -2317.651} C_VEL
LIN {X 0,Y 572.979,Z 279.813,A -85,B 0,C 180,E1 -2319.163,E2 -2319.163} C_VEL
LIN {X 0,Y 572.955,Z 282.45,A -85,B 0,C 180,E1 -2321.402,E2 -2321.402} C_VEL
LIN {X 0,Y 572.94,Z 285.087,A -85,B 0,C 180,E1 -2323.613,E2 -2323.613} C_VEL
LIN {X 0,Y 572.975,Z 288.603,A -85,B 0,C 180,E1 -2326.523,E2 -2326.523} C_VEL
LIN {X 0,Y 572.987,Z 289.894,A -85,B 0,C 180,E1 -2327.583,E2 -2327.583} C_VEL
LIN {X 0,Y 573.866,Z 296.399,A -85,B 0,C 180,E1 -2327.759,E2 -2327.759} C_VEL
LIN {X 0,Y 573.696,Z 309.748,A -85,B 0,C 180,E1 -2328.159,E2 -2328.159} C_VEL
LIN {X 0,Y 573.582,Z 320.583,A -85,B 0,C 180,E1 -2328.614,E2 -2328.614} C_VEL
LIN {X 0,Y 573.511,Z 330.701,A -85,B 0,C 180,E1 -2329.153,E2 -2329.153} C_VEL
LIN {X 0,Y 573.468,Z 340.043,A -85,B 0,C 180,E1 -2329.764,E2 -2329.764} C_VEL
LIN {X 0,Y 573.309,Z 349.056,A -85,B 0,C 180,E1 -2330.474,E2 -2330.474} C_VEL
LIN {X 0,Y 573.237,Z 358.373,A -85,B 0,C 180,E1 -2331.362,E2 -2331.362} C_VEL
LIN {X 0,Y 573.143,Z 367.361,A -85,B 0,C 180,E1 -2332.425,E2 -2332.425} C_VEL
LIN {X 0,Y 573.09,Z 373.912,A -85,B 0,C 180,E1 -2333.382,E2 -2333.382} C_VEL
LIN {X 0,Y 573.071,Z 379.438,A -85,B 0,C 180,E1 -2334.37,E2 -2334.37} C_VEL
LIN {X 0,Y 573.028,Z 384.165,A -85,B 0,C 180,E1 -2335.428,E2 -2335.428} C_VEL
LIN {X 0,Y 573.022,Z 387.792,A -85,B 0,C 180,E1 -2336.484,E2 -2336.484} C_VEL
LIN {X 0,Y 572.959,Z 389.689,A -85,B 0,C 180,E1 -2337.188,E2 -2337.188} C_VEL
LIN {X 0,Y 572.94,Z 391.136,A -85,B 0,C 180,E1 -2337.891,E2 -2337.891} C_VEL
LIN {X 0,Y 572.941,Z 392.755,A -85,B 0,C 180,E1 -2339.297,E2 -2339.297} C_VEL
LIN {X 0,Y 572.939,Z 392.996,A -85,B 0,C 180,E1 -2340,E2 -2340} C_VEL
LIN {X 0,Y 572.947,Z 392.227,A -85,B 0,C 180,E1 -2341.406,E2 -2341.406} C_VEL
LIN {X 0,Y 572.94,Z 391.279,A -85,B 0,C 180,E1 -2342.109,E2 -2342.109} C_VEL
LIN {X 0,Y 572.959,Z 389.874,A -85,B 0,C 180,E1 -2342.812,E2 -2342.812} C_VEL
LIN {X 0,Y 573.015,Z 387.004,A -85,B 0,C 180,E1 -2343.868,E2 -2343.868} C_VEL
LIN {X 0,Y 572.962,Z 383.117,A -85,B 0,C 180,E1 -2344.926,E2 -2344.926} C_VEL
LIN {X 0,Y 573.072,Z 378.097,A -85,B 0,C 180,E1 -2345.984,E2 -2345.984} C_VEL
LIN {X 0,Y 573.113,Z 370.536,A -85,B 0,C 180,E1 -2347.221,E2 -2347.221} C_VEL
LIN {X 0,Y 573.169,Z 363.826,A -85,B 0,C 180,E1 -2348.106,E2 -2348.106} C_VEL
LIN {X 0,Y 573.251,Z 355.737,A -85,B 0,C 180,E1 -2348.993,E2 -2348.993} C_VEL
LIN {X 0,Y 573.329,Z 346.965,A -85,B 0,C 180,E1 -2349.793,E2 -2349.793} C_VEL
LIN {X 0,Y 573.462,Z 336.257,A -85,B 0,C 180,E1 -2350.593,E2 -2350.593} C_VEL
LIN {X 0,Y 573.551,Z 324.052,A -85,B 0,C 180,E1 -2351.306,E2 -2351.306} C_VEL
LIN {X 0,Y 573.667,Z 312.485,A -85,B 0,C 180,E1 -2351.824,E2 -2351.824} C_VEL
LIN {X 0,Y 573.77,Z 301.328,A -85,B 0,C 180,E1 -2352.198,E2 -2352.198} C_VEL
LIN {X 0,Y 573.659,Z 294.448,A -85,B 0,C 180,E1 -2352.38,E2 -2352.38} C_VEL
LIN {X 0,Y 572.945,Z 289.893,A -85,B 0,C 180,E1 -2352.508,E2 -2352.508} C_VEL
LIN {X 0,Y 572.93,Z 286.953,A -85,B 0,C 180,E1 -2354.928,E2 -2354.928} C_VEL
LIN {X 0,Y 572.934,Z 283.436,A -85,B 0,C 180,E1 -2357.859,E2 -2357.859} C_VEL
LIN {X 0,Y 572.962,Z 280.347,A -85,B 0,C 180,E1 -2360.472,E2 -2360.472} C_VEL
LIN {X 0,Y 572.304,Z 279.767,A -85,B 0,C 180,E1 -2361.055,E2 -2361.055} C_VEL
LIN {X 0,Y 569.459,Z 279.212,A -85,B 0,C 180,E1 -2362.006,E2 -2362.006} C_VEL
LIN {X 0,Y 567.072,Z 279.031,A -85,B 0,C 180,E1 -2362.772,E2 -2362.772} C_VEL
LIN {X 0,Y 566.076,Z 278.986,A -85,B 0,C 180,E1 -2363.364,E2 -2363.364} C_VEL
LIN {X 0,Y 566.011,Z 278.981,A -85,B 0,C 180,E1 -2363.564,E2 -2363.564} C_VEL
LIN {X 0,Y 566.198,Z 278.951,A -85,B 0,C 180,E1 -2365.75,E2 -2365.75} C_VEL
LIN {X 0,Y 566.207,Z 278.954,A -85,B 0,C 180,E1 -2368.202,E2 -2368.202} C_VEL
LIN {X 0,Y 566.191,Z 278.953,A -85,B 0,C 180,E1 -2371.076,E2 -2371.076} C_VEL
LIN {X 0,Y 566.215,Z 278.951,A -85,B 0,C 180,E1 -2373.734,E2 -2373.734} C_VEL
LIN {X 0,Y 566.203,Z 278.956,A -85,B 0,C 180,E1 -2376.57,E2 -2376.57} C_VEL
LIN {X 0,Y 566.219,Z 278.952,A -85,B 0,C 180,E1 -2379.686,E2 -2379.686} C_VEL
LIN {X 0,Y 566.213,Z 278.959,A -85,B 0,C 180,E1 -2382.088,E2 -2382.088} C_VEL
LIN {X 0,Y 566.177,Z 278.955,A -85,B 0,C 180,E1 -2385.036,E2 -2385.036} C_VEL
LIN {X 0,Y 566.213,Z 278.958,A -85,B 0,C 180,E1 -2387.912,E2 -2387.912} C_VEL
LIN {X 0,Y 566.218,Z 278.95,A -85,B 0,C 180,E1 -2390.726,E2 -2390.726} C_VEL
LIN {X 0,Y 566.187,Z 278.96,A -85,B 0,C 180,E1 -2393.788,E2 -2393.788} C_VEL
LIN {X 0,Y 566.103,Z 279.08,A -85,B 0,C 180,E1 -2395.822,E2 -2395.822} C_VEL
LIN {X 0,Y 566.033,Z 284.284,A -85,B 0,C 180,E1 -2398.568,E2 -2398.568} C_VEL
LIN {X 0,Y 565.978,Z 288.692,A -85,B 0,C 180,E1 -2401.035,E2 -2401.035} C_VEL
LIN {X 0,Y 566.019,Z 293.024,A -85,B 0,C 180,E1 -2403.449,E2 -2403.449} C_VEL
LIN {X 0,Y 565.968,Z 297.287,A -85,B 0,C 180,E1 -2405.809,E2 -2405.809} C_VEL
LIN {X 0,Y 565.968,Z 302.336,A -85,B 0,C 180,E1 -2408.643,E2 -2408.643} C_VEL
LIN {X 0,Y 565.955,Z 306.867,A -85,B 0,C 180,E1 -2411.164,E2 -2411.164} C_VEL
LIN {X 0,Y 565.883,Z 312.396,A -85,B 0,C 180,E1 -2414.143,E2 -2414.143} C_VEL
LIN {X 0,Y 565.892,Z 316.544,A -85,B 0,C 180,E1 -2416.351,E2 -2416.351} C_VEL
LIN {X 0,Y 565.91,Z 318.663,A -85,B 0,C 180,E1 -2417.425,E2 -2417.425} C_VEL
LIN {X 0,Y 566.911,Z 325.394,A -85,B 0,C 180,E1 -2417.584,E2 -2417.584} C_VEL
LIN {X 0,Y 566.782,Z 337.074,A -85,B 0,C 180,E1 -2417.922,E2 -2417.922} C_VEL
LIN {X 0,Y 566.657,Z 347.721,A -85,B 0,C 180,E1 -2418.341,E2 -2418.341} C_VEL
LIN {X 0,Y 566.536,Z 358.159,A -85,B 0,C 180,E1 -2418.869,E2 -2418.869} C_VEL
LIN {X 0,Y 566.442,Z 368.851,A -85,B 0,C 180,E1 -2419.545,E2 -2419.545} C_VEL
LIN {X 0,Y 566.301,Z 379.134,A -85,B 0,C 180,E1 -2420.355,E2 -2420.355} C_VEL
LIN {X 0,Y 566.167,Z 388.335,A -85,B 0,C 180,E1 -2421.253,E2 -2421.253} C_VEL
LIN {X 0,Y 566.095,Z 395.943,A -85,B 0,C 180,E1 -2422.151,E2 -2422.151} C_VEL
LIN {X 0,Y 566.021,Z 402.805,A -85,B 0,C 180,E1 -2423.127,E2 -2423.127} C_VEL
LIN {X 0,Y 566,Z 409.455,A -85,B 0,C 180,E1 -2424.299,E2 -2424.299} C_VEL
LIN {X 0,Y 565.932,Z 414.204,A -85,B 0,C 180,E1 -2425.37,E2 -2425.37} C_VEL
LIN {X 0,Y 565.927,Z 417.838,A -85,B 0,C 180,E1 -2426.44,E2 -2426.44} C_VEL
LIN {X 0,Y 565.877,Z 419.669,A -85,B 0,C 180,E1 -2427.152,E2 -2427.152} C_VEL
LIN {X 0,Y 565.845,Z 422.144,A -85,B 0,C 180,E1 -2428.577,E2 -2428.577} C_VEL
LIN {X 0,Y 565.841,Z 422.751,A -85,B 0,C 180,E1 -2429.288,E2 -2429.288} C_VEL
LIN {X 0,Y 565.841,Z 422.81,A -85,B 0,C 180,E1 -2430.712,E2 -2430.712} C_VEL
LIN {X 0,Y 565.846,Z 422.243,A -85,B 0,C 180,E1 -2431.423,E2 -2431.423} C_VEL
LIN {X 0,Y 565.878,Z 419.892,A -85,B 0,C 180,E1 -2432.848,E2 -2432.848} C_VEL
LIN {X 0,Y 565.926,Z 417.015,A -85,B 0,C 180,E1 -2433.916,E2 -2433.916} C_VEL
LIN {X 0,Y 565.878,Z 413.103,A -85,B 0,C 180,E1 -2434.987,E2 -2434.987} C_VEL
LIN {X 0,Y 565.991,Z 408.052,A -85,B 0,C 180,E1 -2436.059,E2 -2436.059} C_VEL
LIN {X 0,Y 566.032,Z 401.717,A -85,B 0,C 180,E1 -2437.132,E2 -2437.132} C_VEL
LIN {X 0,Y 566.128,Z 393.87,A -85,B 0,C 180,E1 -2438.208,E2 -2438.208} C_VEL
LIN {X 0,Y 566.249,Z 383.945,A -85,B 0,C 180,E1 -2439.285,E2 -2439.285} C_VEL
LIN {X 0,Y 566.401,Z 374.754,A -85,B 0,C 180,E1 -2440.094,E2 -2440.094} C_VEL
LIN {X 0,Y 566.464,Z 364.976,A -85,B 0,C 180,E1 -2440.805,E2 -2440.805} C_VEL
LIN {X 0,Y 566.574,Z 354.064,A -85,B 0,C 180,E1 -2441.448,E2 -2441.448} C_VEL
LIN {X 0,Y 566.748,Z 341.293,A -85,B 0,C 180,E1 -2442.02,E2 -2442.02} C_VEL
LIN {X 0,Y 566.87,Z 328.862,A -85,B 0,C 180,E1 -2442.417,E2 -2442.417} C_VEL
LIN {X 0,Y 566.709,Z 323.446,A -85,B 0,C 180,E1 -2442.558,E2 -2442.558} C_VEL
LIN {X 0,Y 565.894,Z 318.596,A -85,B 0,C 180,E1 -2442.667,E2 -2442.667} C_VEL
LIN {X 0,Y 565.914,Z 313.948,A -85,B 0,C 180,E1 -2445.117,E2 -2445.117} C_VEL
LIN {X 0,Y 565.898,Z 308.415,A -85,B 0,C 180,E1 -2448.088,E2 -2448.088} C_VEL
LIN {X 0,Y 565.933,Z 304.272,A -85,B 0,C 180,E1 -2450.348,E2 -2450.348} C_VEL
LIN {X 0,Y 566.005,Z 299.121,A -85,B 0,C 180,E1 -2453.241,E2 -2453.241} C_VEL
LIN {X 0,Y 566.013,Z 294.629,A -85,B 0,C 180,E1 -2455.759,E2 -2455.759} C_VEL
LIN {X 0,Y 566.002,Z 290.297,A -85,B 0,C 180,E1 -2458.163,E2 -2458.163} C_VEL
LIN {X 0,Y 566.046,Z 285.134,A -85,B 0,C 180,E1 -2461.051,E2 -2461.051} C_VEL
LIN {X 0,Y 566.091,Z 279.691,A -85,B 0,C 180,E1 -2463.964,E2 -2463.964} C_VEL
LIN {X 0,Y 566.153,Z 278.967,A -85,B 0,C 180,E1 -2464.39,E2 -2464.39} C_VEL
LIN {X 0,Y 566.195,Z 278.959,A -85,B 0,C 180,E1 -2467.461,E2 -2467.461} C_VEL
LIN {X 0,Y 566.212,Z 278.956,A -85,B 0,C 180,E1 -2470.199,E2 -2470.199} C_VEL
LIN {X 0,Y 566.204,Z 278.957,A -85,B 0,C 180,E1 -2473.054,E2 -2473.054} C_VEL
LIN {X 0,Y 566.197,Z 278.959,A -85,B 0,C 180,E1 -2476.049,E2 -2476.049} C_VEL
LIN {X 0,Y 566.206,Z 278.957,A -85,B 0,C 180,E1 -2479.215,E2 -2479.215} C_VEL
LIN {X 0,Y 566.188,Z 278.96,A -85,B 0,C 180,E1 -2481.637,E2 -2481.637} C_VEL
LIN {X 0,Y 566.151,Z 278.964,A -85,B 0,C 180,E1 -2484.307,E2 -2484.307} C_VEL
LIN {X 0,Y 566.089,Z 279.105,A -85,B 0,C 180,E1 -2485.928,E2 -2485.928} C_VEL
LIN {X 0,Y 566.033,Z 284.766,A -85,B 0,C 180,E1 -2488.951,E2 -2488.951} C_VEL
LIN {X 0,Y 565.999,Z 290.095,A -85,B 0,C 180,E1 -2491.846,E2 -2491.846} C_VEL
LIN {X 0,Y 566.012,Z 294.473,A -85,B 0,C 180,E1 -2494.241,E2 -2494.241} C_VEL
LIN {X 0,Y 566.005,Z 298.991,A -85,B 0,C 180,E1 -2496.759,E2 -2496.759} C_VEL
LIN {X 0,Y 565.931,Z 304.106,A -85,B 0,C 180,E1 -2499.652,E2 -2499.652} C_VEL
LIN {X 0,Y 565.902,Z 308.249,A -85,B 0,C 180,E1 -2501.912,E2 -2501.912} C_VEL
LIN {X 0,Y 565.915,Z 313.779,A -85,B 0,C 180,E1 -2504.883,E2 -2504.883} C_VEL
LIN {X 0,Y 565.91,Z 318.731,A -85,B 0,C 180,E1 -2507.425,E2 -2507.425} C_VEL
LIN {X 0,Y 566.902,Z 326.239,A -85,B 0,C 180,E1 -2507.606,E2 -2507.606} C_VEL
LIN {X 0,Y 566.8,Z 337.117,A -85,B 0,C 180,E1 -2507.922,E2 -2507.922} C_VEL
LIN {X 0,Y 566.663,Z 349.624,A -85,B 0,C 180,E1 -2508.423,E2 -2508.423} C_VEL
LIN {X 0,Y 566.554,Z 360.945,A -85,B 0,C 180,E1 -2509.03,E2 -2509.03} C_VEL
LIN {X 0,Y 566.426,Z 371.265,A -85,B 0,C 180,E1 -2509.726,E2 -2509.726} C_VEL
LIN {X 0,Y 566.302,Z 379.072,A -85,B 0,C 180,E1 -2510.355,E2 -2510.355} C_VEL
LIN {X 0,Y 566.167,Z 388.321,A -85,B 0,C 180,E1 -2511.253,E2 -2511.253} C_VEL
LIN {X 0,Y 566.095,Z 395.956,A -85,B 0,C 180,E1 -2512.151,E2 -2512.151} C_VEL
LIN {X 0,Y 566.019,Z 402.835,A -85,B 0,C 180,E1 -2513.127,E2 -2513.127} C_VEL
LIN {X 0,Y 566.002,Z 409.468,A -85,B 0,C 180,E1 -2514.299,E2 -2514.299} C_VEL
LIN {X 0,Y 565.933,Z 414.208,A -85,B 0,C 180,E1 -2515.37,E2 -2515.37} C_VEL
LIN {X 0,Y 565.927,Z 417.836,A -85,B 0,C 180,E1 -2516.44,E2 -2516.44} C_VEL
LIN {X 0,Y 565.877,Z 419.687,A -85,B 0,C 180,E1 -2517.152,E2 -2517.152} C_VEL
LIN {X 0,Y 565.845,Z 422.136,A -85,B 0,C 180,E1 -2518.577,E2 -2518.577} C_VEL
LIN {X 0,Y 565.841,Z 422.759,A -85,B 0,C 180,E1 -2519.288,E2 -2519.288} C_VEL
LIN {X 0,Y 565.841,Z 422.803,A -85,B 0,C 180,E1 -2520.712,E2 -2520.712} C_VEL
LIN {X 0,Y 565.846,Z 422.245,A -85,B 0,C 180,E1 -2521.423,E2 -2521.423} C_VEL
LIN {X 0,Y 565.878,Z 419.888,A -85,B 0,C 180,E1 -2522.848,E2 -2522.848} C_VEL
LIN {X 0,Y 565.926,Z 417.013,A -85,B 0,C 180,E1 -2523.916,E2 -2523.916} C_VEL
LIN {X 0,Y 565.878,Z 413.104,A -85,B 0,C 180,E1 -2524.987,E2 -2524.987} C_VEL
LIN {X 0,Y 565.994,Z 408.053,A -85,B 0,C 180,E1 -2526.059,E2 -2526.059} C_VEL
LIN {X 0,Y 566.032,Z 401.711,A -85,B 0,C 180,E1 -2527.132,E2 -2527.132} C_VEL
LIN {X 0,Y 566.128,Z 393.861,A -85,B 0,C 180,E1 -2528.208,E2 -2528.208} C_VEL
LIN {X 0,Y 566.247,Z 383.969,A -85,B 0,C 180,E1 -2529.285,E2 -2529.285} C_VEL
LIN {X 0,Y 566.398,Z 374.76,A -85,B 0,C 180,E1 -2530.094,E2 -2530.094} C_VEL
LIN {X 0,Y 566.461,Z 364.975,A -85,B 0,C 180,E1 -2530.804,E2 -2530.804} C_VEL
LIN {X 0,Y 566.583,Z 355.773,A -85,B 0,C 180,E1 -2531.352,E2 -2531.352} C_VEL
LIN {X 0,Y 566.668,Z 345.361,A -85,B 0,C 180,E1 -2531.853,E2 -2531.853} C_VEL
LIN {X 0,Y 566.871,Z 333.028,A -85,B 0,C 180,E1 -2532.303,E2 -2532.303} C_VEL
LIN {X 0,Y 566.763,Z 323.928,A -85,B 0,C 180,E1 -2532.545,E2 -2532.545} C_VEL
LIN {X 0,Y 565.895,Z 318.529,A -85,B 0,C 180,E1 -2532.689,E2 -2532.689} C_VEL
LIN {X 0,Y 565.914,Z 313.948,A -85,B 0,C 180,E1 -2535.117,E2 -2535.117} C_VEL
LIN {X 0,Y 565.898,Z 308.415,A -85,B 0,C 180,E1 -2538.088,E2 -2538.088} C_VEL
LIN {X 0,Y 565.932,Z 304.27,A -85,B 0,C 180,E1 -2540.348,E2 -2540.348} C_VEL
LIN {X 0,Y 566.015,Z 299.149,A -85,B 0,C 180,E1 -2543.244,E2 -2543.244} C_VEL
LIN {X 0,Y 566.005,Z 294.348,A -85,B 0,C 180,E1 -2545.759,E2 -2545.759} C_VEL
LIN {X 0,Y 565.964,Z 289.487,A -85,B 0,C 180,E1 -2548.156,E2 -2548.156} C_VEL
LIN {X 0,Y 565.889,Z 283.092,A -85,B 0,C 180,E1 -2551.025,E2 -2551.025} C_VEL
LIN {X 0,Y 565.936,Z 278.994,A -85,B 0,C 180,E1 -2552.72,E2 -2552.72} C_VEL
LIN {X 0,Y 566.173,Z 278.964,A -85,B 0,C 180,E1 -2554.988,E2 -2554.988} C_VEL
LIN {X 0,Y 566.199,Z 278.959,A -85,B 0,C 180,E1 -2557.461,E2 -2557.461} C_VEL
LIN {X 0,Y 566.209,Z 278.958,A -85,B 0,C 180,E1 -2560.199,E2 -2560.199} C_VEL
LIN {X 0,Y 566.197,Z 278.961,A -85,B 0,C 180,E1 -2563.055,E2 -2563.055} C_VEL
LIN {X 0,Y 566.2,Z 278.957,A -85,B 0,C 180,E1 -2566.049,E2 -2566.049} C_VEL
LIN {X 0,Y 566.206,Z 278.958,A -85,B 0,C 180,E1 -2569.215,E2 -2569.215} C_VEL
LIN {X 0,Y 566.184,Z 278.96,A -85,B 0,C 180,E1 -2571.636,E2 -2571.636} C_VEL
LIN {X 0,Y 566.246,Z 279.146,A -85,B 0,C 180,E1 -2572.737,E2 -2572.737} C_VEL
LIN {X 0,Y 567.196,Z 284.737,A -85,B 0,C 180,E1 -2574.383,E2 -2574.383} C_VEL
LIN {X 0,Y 566.986,Z 293.946,A -85,B 0,C 180,E1 -2576.948,E2 -2576.948} C_VEL
LIN {X 0,Y 566.846,Z 303.154,A -85,B 0,C 180,E1 -2579.447,E2 -2579.447} C_VEL
LIN {X 0,Y 566.696,Z 313.897,A -85,B 0,C 180,E1 -2582.286,E2 -2582.286} C_VEL
LIN {X 0,Y 566.538,Z 324.641,A -85,B 0,C 180,E1 -2585.053,E2 -2585.053} C_VEL
LIN {X 0,Y 566.414,Z 335.384,A -85,B 0,C 180,E1 -2587.763,E2 -2587.763} C_VEL
LIN {X 0,Y 566.319,Z 346.803,A -85,B 0,C 180,E1 -2590.589,E2 -2590.589} C_VEL
LIN {X 0,Y 566.196,Z 358.405,A -85,B 0,C 180,E1 -2593.412,E2 -2593.412} C_VEL
LIN {X 0,Y 566.086,Z 370.683,A -85,B 0,C 180,E1 -2596.356,E2 -2596.356} C_VEL
LIN {X 0,Y 566.061,Z 374.712,A -85,B 0,C 180,E1 -2597.314,E2 -2597.314} C_VEL
LIN {X 0,Y 566.957,Z 381.227,A -85,B 0,C 180,E1 -2597.448,E2 -2597.448} C_VEL
LIN {X 0,Y 566.834,Z 394.495,A -85,B 0,C 180,E1 -2597.787,E2 -2597.787} C_VEL
LIN {X 0,Y 566.688,Z 406.318,A -85,B 0,C 180,E1 -2598.228,E2 -2598.228} C_VEL
LIN {X 0,Y 566.532,Z 418.967,A -85,B 0,C 180,E1 -2598.867,E2 -2598.867} C_VEL
LIN {X 0,Y 566.434,Z 430.746,A -85,B 0,C 180,E1 -2599.636,E2 -2599.636} C_VEL
LIN {X 0,Y 566.301,Z 439.646,A -85,B 0,C 180,E1 -2600.355,E2 -2600.355} C_VEL
LIN {X 0,Y 566.166,Z 448.787,A -85,B 0,C 180,E1 -2601.253,E2 -2601.253} C_VEL
LIN {X 0,Y 566.081,Z 457.69,A -85,B 0,C 180,E1 -2602.33,E2 -2602.33} C_VEL
LIN {X 0,Y 565.967,Z 464.955,A -85,B 0,C 180,E1 -2603.422,E2 -2603.422} C_VEL
LIN {X 0,Y 566.004,Z 469.68,A -85,B 0,C 180,E1 -2604.299,E2 -2604.299} C_VEL
LIN {X 0,Y 565.933,Z 474.371,A -85,B 0,C 180,E1 -2605.37,E2 -2605.37} C_VEL
LIN {X 0,Y 565.927,Z 477.956,A -85,B 0,C 180,E1 -2606.44,E2 -2606.44} C_VEL
LIN {X 0,Y 565.878,Z 479.809,A -85,B 0,C 180,E1 -2607.152,E2 -2607.152} C_VEL
LIN {X 0,Y 565.841,Z 481.2,A -85,B 0,C 180,E1 -2607.865,E2 -2607.865} C_VEL
LIN {X 0,Y 565.841,Z 482.784,A -85,B 0,C 180,E1 -2609.288,E2 -2609.288} C_VEL
LIN {X 0,Y 565.839,Z 483,A -85,B 0,C 180,E1 -2610,E2 -2610} C_VEL
LIN {X 0,Y 565.846,Z 482.185,A -85,B 0,C 180,E1 -2611.423,E2 -2611.423} C_VEL
LIN {X 0,Y 565.841,Z 481.201,A -85,B 0,C 180,E1 -2612.135,E2 -2612.135} C_VEL
LIN {X 0,Y 565.878,Z 479.81,A -85,B 0,C 180,E1 -2612.848,E2 -2612.848} C_VEL
LIN {X 0,Y 565.926,Z 476.896,A -85,B 0,C 180,E1 -2613.916,E2 -2613.916} C_VEL
LIN {X 0,Y 565.878,Z 472.949,A -85,B 0,C 180,E1 -2614.987,E2 -2614.987} C_VEL
LIN {X 0,Y 566.002,Z 467.866,A -85,B 0,C 180,E1 -2616.059,E2 -2616.059} C_VEL
LIN {X 0,Y 566.04,Z 461.469,A -85,B 0,C 180,E1 -2617.132,E2 -2617.132} C_VEL
LIN {X 0,Y 566.134,Z 453.478,A -85,B 0,C 180,E1 -2618.208,E2 -2618.208} C_VEL
LIN {X 0,Y 566.229,Z 445.336,A -85,B 0,C 180,E1 -2619.106,E2 -2619.106} C_VEL
LIN {X 0,Y 566.344,Z 435.401,A -85,B 0,C 180,E1 -2620.005,E2 -2620.005} C_VEL
LIN {X 0,Y 566.501,Z 424.327,A -85,B 0,C 180,E1 -2620.805,E2 -2620.805} C_VEL
LIN {X 0,Y 566.573,Z 413.177,A -85,B 0,C 180,E1 -2621.448,E2 -2621.448} C_VEL
LIN {X 0,Y 566.736,Z 400.987,A -85,B 0,C 180,E1 -2621.988,E2 -2621.988} C_VEL
LIN {X 0,Y 566.883,Z 388.176,A -85,B 0,C 180,E1 -2622.394,E2 -2622.394} C_VEL
LIN {X 0,Y 566.759,Z 379.229,A -85,B 0,C 180,E1 -2622.596,E2 -2622.596} C_VEL
LIN {X 0,Y 566.061,Z 374.712,A -85,B 0,C 180,E1 -2622.686,E2 -2622.686} C_VEL
LIN {X 0,Y 566.133,Z 363.009,A -85,B 0,C 180,E1 -2625.48,E2 -2625.48} C_VEL
LIN {X 0,Y 566.239,Z 352.266,A -85,B 0,C 180,E1 -2628.077,E2 -2628.077} C_VEL
LIN {X 0,Y 566.339,Z 341.523,A -85,B 0,C 180,E1 -2630.712,E2 -2630.712} C_VEL
LIN {X 0,Y 566.52,Z 329.245,A -85,B 0,C 180,E1 -2633.777,E2 -2633.777} C_VEL
LIN {X 0,Y 566.616,Z 317.653,A -85,B 0,C 180,E1 -2636.741,E2 -2636.741} C_VEL
LIN {X 0,Y 566.8,Z 307.758,A -85,B 0,C 180,E1 -2639.326,E2 -2639.326} C_VEL
LIN {X 0,Y 566.961,Z 297.015,A -85,B 0,C 180,E1 -2642.21,E2 -2642.21} C_VEL
LIN {X 0,Y 567.12,Z 287.807,A -85,B 0,C 180,E1 -2644.754,E2 -2644.754} C_VEL
LIN {X 0,Y 567.054,Z 283.574,A -85,B 0,C 180,E1 -2645.953,E2 -2645.953} C_VEL
LIN {X 0,Y 566.188,Z 278.962,A -85,B 0,C 180,E1 -2647.265,E2 -2647.265} C_VEL
LIN {X 0,Y 566.207,Z 278.955,A -85,B 0,C 180,E1 -2650.199,E2 -2650.199} C_VEL
LIN {X 0,Y 566.182,Z 278.96,A -85,B 0,C 180,E1 -2653.056,E2 -2653.056} C_VEL
LIN {X 0,Y 566.195,Z 278.957,A -85,B 0,C 180,E1 -2656.049,E2 -2656.049} C_VEL
LIN {X 0,Y 566.206,Z 278.953,A -85,B 0,C 180,E1 -2659.215,E2 -2659.215} C_VEL
LIN {X 0,Y 566.189,Z 278.957,A -85,B 0,C 180,E1 -2661.637,E2 -2661.637} C_VEL
LIN {X 0,Y 566.165,Z 278.962,A -85,B 0,C 180,E1 -2664.308,E2 -2664.308} C_VEL
LIN {X 0,Y 566.223,Z 278.95,A -85,B 0,C 180,E1 -2666.898,E2 -2666.898} C_VEL
LIN {X 0,Y 566.184,Z 278.96,A -85,B 0,C 180,E1 -2669.407,E2 -2669.407} C_VEL
LIN {X 0,Y 566.215,Z 278.957,A -85,B 0,C 180,E1 -2671.857,E2 -2671.857} C_VEL
LIN {X 0,Y 566.202,Z 278.954,A -85,B 0,C 180,E1 -2674.25,E2 -2674.25} C_VEL
LIN {X 0,Y 566.021,Z 278.982,A -85,B 0,C 180,E1 -2676.755,E2 -2676.755} C_VEL
LIN {X 0,Y 565.93,Z 278.995,A -85,B 0,C 180,E1 -2677.358,E2 -2677.358} C_VEL
LIN {X 0,Y 565.908,Z 280.949,A -85,B 0,C 180,E1 -2679.651,E2 -2679.651} C_VEL
LIN {X 0,Y 565.858,Z 283.33,A -85,B 0,C 180,E1 -2681.91,E2 -2681.91} C_VEL
LIN {X 0,Y 565.831,Z 286.845,A -85,B 0,C 180,E1 -2684.88,E2 -2684.88} C_VEL
LIN {X 0,Y 565.86,Z 289.894,A -85,B 0,C 180,E1 -2687.424,E2 -2687.424} C_VEL
LIN {X 0,Y 566.899,Z 297.348,A -85,B 0,C 180,E1 -2687.629,E2 -2687.629} C_VEL
LIN {X 0,Y 566.726,Z 310.876,A -85,B 0,C 180,E1 -2688.057,E2 -2688.057} C_VEL
LIN {X 0,Y 566.574,Z 322.199,A -85,B 0,C 180,E1 -2688.552,E2 -2688.552} C_VEL
LIN {X 0,Y 566.512,Z 332.286,A -85,B 0,C 180,E1 -2689.115,E2 -2689.115} C_VEL
LIN {X 0,Y 566.416,Z 342.502,A -85,B 0,C 180,E1 -2689.816,E2 -2689.816} C_VEL
LIN {X 0,Y 566.276,Z 353.066,A -85,B 0,C 180,E1 -2690.715,E2 -2690.715} C_VEL
LIN {X 0,Y 566.154,Z 361.565,A -85,B 0,C 180,E1 -2691.613,E2 -2691.613} C_VEL
LIN {X 0,Y 566.057,Z 368.63,A -85,B 0,C 180,E1 -2692.509,E2 -2692.509} C_VEL
LIN {X 0,Y 565.969,Z 375.575,A -85,B 0,C 180,E1 -2693.583,E2 -2693.583} C_VEL
LIN {X 0,Y 565.937,Z 381.152,A -85,B 0,C 180,E1 -2694.656,E2 -2694.656} C_VEL
LIN {X 0,Y 565.959,Z 385.53,A -85,B 0,C 180,E1 -2695.727,E2 -2695.727} C_VEL
LIN {X 0,Y 565.877,Z 389.684,A -85,B 0,C 180,E1 -2697.152,E2 -2697.152} C_VEL
LIN {X 0,Y 565.841,Z 391.136,A -85,B 0,C 180,E1 -2697.865,E2 -2697.865} C_VEL
LIN {X 0,Y 565.841,Z 392.748,A -85,B 0,C 180,E1 -2699.288,E2 -2699.288} C_VEL
LIN {X 0,Y 565.839,Z 392.996,A -85,B 0,C 180,E1 -2700,E2 -2700} C_VEL
LIN {X 0,Y 565.846,Z 392.222,A -85,B 0,C 180,E1 -2701.423,E2 -2701.423} C_VEL
LIN {X 0,Y 565.841,Z 391.279,A -85,B 0,C 180,E1 -2702.135,E2 -2702.135} C_VEL
LIN {X 0,Y 565.927,Z 388.051,A -85,B 0,C 180,E1 -2703.56,E2 -2703.56} C_VEL
LIN {X 0,Y 565.933,Z 384.505,A -85,B 0,C 180,E1 -2704.63,E2 -2704.63} C_VEL
LIN {X 0,Y 565.999,Z 379.862,A -85,B 0,C 180,E1 -2705.701,E2 -2705.701} C_VEL
LIN {X 0,Y 565.996,Z 372.91,A -85,B 0,C 180,E1 -2706.954,E2 -2706.954} C_VEL
LIN {X 0,Y 566.105,Z 365.305,A -85,B 0,C 180,E1 -2708.029,E2 -2708.029} C_VEL
LIN {X 0,Y 566.202,Z 357.501,A -85,B 0,C 180,E1 -2708.926,E2 -2708.926} C_VEL
LIN {X 0,Y 566.309,Z 349.053,A -85,B 0,C 180,E1 -2709.735,E2 -2709.735} C_VEL
LIN {X 0,Y 566.398,Z 340.025,A -85,B 0,C 180,E1 -2710.456,E2 -2710.456} C_VEL
LIN {X 0,Y 566.512,Z 329.845,A -85,B 0,C 180,E1 -2711.123,E2 -2711.123} C_VEL
LIN {X 0,Y 566.672,Z 319.23,A -85,B 0,C 180,E1 -2711.682,E2 -2711.682} C_VEL
LIN {X 0,Y 566.814,Z 305.866,A -85,B 0,C 180,E1 -2712.214,E2 -2712.214} C_VEL
LIN {X 0,Y 566.723,Z 295.311,A -85,B 0,C 180,E1 -2712.514,E2 -2712.514} C_VEL
LIN {X 0,Y 565.86,Z 289.893,A -85,B 0,C 180,E1 -2712.667,E2 -2712.667} C_VEL
LIN {X 0,Y 565.828,Z 286.953,A -85,B 0,C 180,E1 -2715.12,E2 -2715.12} C_VEL
LIN {X 0,Y 565.829,Z 284.315,A -85,B 0,C 180,E1 -2717.343,E2 -2717.343} C_VEL
LIN {X 0,Y 565.853,Z 281.677,A -85,B 0,C 180,E1 -2719.594,E2 -2719.594} C_VEL
LIN {X 0,Y 565.88,Z 279.266,A -85,B 0,C 180,E1 -2721.875,E2 -2721.875} C_VEL
LIN {X 0,Y 566.011,Z 278.981,A -85,B 0,C 180,E1 -2723.564,E2 -2723.564} C_VEL
LIN {X 0,Y 565.399,Z 279.059,A -85,B 0,C 180,E1 -2724.159,E2 -2724.159} C_VEL
LIN {X 0,Y 562.612,Z 279.401,A -85,B 0,C 180,E1 -2725.124,E2 -2725.124} C_VEL
LIN {X 0,Y 560.242,Z 279.694,A -85,B 0,C 180,E1 -2725.901,E2 -2725.901} C_VEL
LIN {X 0,Y 559.237,Z 279.825,A -85,B 0,C 180,E1 -2726.501,E2 -2726.501} C_VEL
LIN {X 0,Y 559.164,Z 279.832,A -85,B 0,C 180,E1 -2726.704,E2 -2726.704} C_VEL
LIN {X 0,Y 559.143,Z 279.831,A -85,B 0,C 180,E1 -2729.354,E2 -2729.354} C_VEL
LIN {X 0,Y 559.169,Z 279.828,A -85,B 0,C 180,E1 -2731.863,E2 -2731.863} C_VEL
LIN {X 0,Y 559.145,Z 279.837,A -85,B 0,C 180,E1 -2734.445,E2 -2734.445} C_VEL
LIN {X 0,Y 559.144,Z 279.831,A -85,B 0,C 180,E1 -2737.108,E2 -2737.108} C_VEL
LIN {X 0,Y 559.165,Z 279.835,A -85,B 0,C 180,E1 -2739.942,E2 -2739.942} C_VEL
LIN {X 0,Y 559.164,Z 279.829,A -85,B 0,C 180,E1 -2742.743,E2 -2742.743} C_VEL
LIN {X 0,Y 559.157,Z 279.837,A -85,B 0,C 180,E1 -2745.761,E2 -2745.761} C_VEL
LIN {X 0,Y 559.17,Z 279.831,A -85,B 0,C 180,E1 -2748.23,E2 -2748.23} C_VEL
LIN {X 0,Y 559.178,Z 279.83,A -85,B 0,C 180,E1 -2751.192,E2 -2751.192} C_VEL
LIN {X 0,Y 559.142,Z 279.838,A -85,B 0,C 180,E1 -2753.789,E2 -2753.789} C_VEL
LIN {X 0,Y 559.044,Z 279.988,A -85,B 0,C 180,E1 -2755.914,E2 -2755.914} C_VEL
LIN {X 0,Y 558.99,Z 285.361,A -85,B 0,C 180,E1 -2758.754,E2 -2758.754} C_VEL
LIN {X 0,Y 558.942,Z 290.498,A -85,B 0,C 180,E1 -2761.662,E2 -2761.662} C_VEL
LIN {X 0,Y 558.973,Z 296.188,A -85,B 0,C 180,E1 -2764.859,E2 -2764.859} C_VEL
LIN {X 0,Y 558.922,Z 301.512,A -85,B 0,C 180,E1 -2767.838,E2 -2767.838} C_VEL
LIN {X 0,Y 558.876,Z 306.918,A -85,B 0,C 180,E1 -2770.916,E2 -2770.916} C_VEL
LIN {X 0,Y 558.791,Z 312.397,A -85,B 0,C 180,E1 -2773.937,E2 -2773.937} C_VEL
LIN {X 0,Y 558.808,Z 316.545,A -85,B 0,C 180,E1 -2776.175,E2 -2776.175} C_VEL
LIN {X 0,Y 558.823,Z 318.644,A -85,B 0,C 180,E1 -2777.263,E2 -2777.263} C_VEL
LIN {X 0,Y 559.963,Z 326.267,A -85,B 0,C 180,E1 -2777.45,E2 -2777.45} C_VEL
LIN {X 0,Y 559.853,Z 337.071,A -85,B 0,C 180,E1 -2777.77,E2 -2777.77} C_VEL
LIN {X 0,Y 559.701,Z 347.715,A -85,B 0,C 180,E1 -2778.194,E2 -2778.194} C_VEL
LIN {X 0,Y 559.58,Z 357.706,A -85,B 0,C 180,E1 -2778.704,E2 -2778.704} C_VEL
LIN {X 0,Y 559.423,Z 368.858,A -85,B 0,C 180,E1 -2779.413,E2 -2779.413} C_VEL
LIN {X 0,Y 559.297,Z 379.139,A -85,B 0,C 180,E1 -2780.233,E2 -2780.233} C_VEL
LIN {X 0,Y 559.141,Z 388.332,A -85,B 0,C 180,E1 -2781.143,E2 -2781.143} C_VEL
LIN {X 0,Y 559.053,Z 395.94,A -85,B 0,C 180,E1 -2782.051,E2 -2782.051} C_VEL
LIN {X 0,Y 558.971,Z 402.399,A -85,B 0,C 180,E1 -2782.977,E2 -2782.977} C_VEL
LIN {X 0,Y 558.912,Z 407.567,A -85,B 0,C 180,E1 -2783.864,E2 -2783.864} C_VEL
LIN {X 0,Y 558.797,Z 412.708,A -85,B 0,C 180,E1 -2784.949,E2 -2784.949} C_VEL
LIN {X 0,Y 558.844,Z 416.705,A -85,B 0,C 180,E1 -2786.034,E2 -2786.034} C_VEL
LIN {X 0,Y 558.799,Z 419.665,A -85,B 0,C 180,E1 -2787.116,E2 -2787.116} C_VEL
LIN {X 0,Y 558.745,Z 422.146,A -85,B 0,C 180,E1 -2788.558,E2 -2788.558} C_VEL
LIN {X 0,Y 558.741,Z 422.751,A -85,B 0,C 180,E1 -2789.279,E2 -2789.279} C_VEL
LIN {X 0,Y 558.741,Z 422.809,A -85,B 0,C 180,E1 -2790.721,E2 -2790.721} C_VEL
LIN {X 0,Y 558.746,Z 422.241,A -85,B 0,C 180,E1 -2791.442,E2 -2791.442} C_VEL
LIN {X 0,Y 558.8,Z 419.886,A -85,B 0,C 180,E1 -2792.884,E2 -2792.884} C_VEL
LIN {X 0,Y 558.844,Z 417.006,A -85,B 0,C 180,E1 -2793.966,E2 -2793.966} C_VEL
LIN {X 0,Y 558.798,Z 413.092,A -85,B 0,C 180,E1 -2795.051,E2 -2795.051} C_VEL
LIN {X 0,Y 558.911,Z 408.04,A -85,B 0,C 180,E1 -2796.136,E2 -2796.136} C_VEL
LIN {X 0,Y 558.975,Z 401.704,A -85,B 0,C 180,E1 -2797.223,E2 -2797.223} C_VEL
LIN {X 0,Y 559.091,Z 393.866,A -85,B 0,C 180,E1 -2798.312,E2 -2798.312} C_VEL
LIN {X 0,Y 559.224,Z 383.929,A -85,B 0,C 180,E1 -2799.403,E2 -2799.403} C_VEL
LIN {X 0,Y 559.351,Z 375.866,A -85,B 0,C 180,E1 -2800.131,E2 -2800.131} C_VEL
LIN {X 0,Y 559.465,Z 366.141,A -85,B 0,C 180,E1 -2800.861,E2 -2800.861} C_VEL
LIN {X 0,Y 559.562,Z 356.491,A -85,B 0,C 180,E1 -2801.455,E2 -2801.455} C_VEL
LIN {X 0,Y 559.758,Z 345.356,A -85,B 0,C 180,E1 -2802.002,E2 -2802.002} C_VEL
LIN {X 0,Y 559.926,Z 331.43,A -85,B 0,C 180,E1 -2802.505,E2 -2802.505} C_VEL
LIN {X 0,Y 559.786,Z 324.41,A -85,B 0,C 180,E1 -2802.692,E2 -2802.692} C_VEL
LIN {X 0,Y 558.794,Z 318.571,A -85,B 0,C 180,E1 -2802.83,E2 -2802.83} C_VEL
LIN {X 0,Y 558.827,Z 313.946,A -85,B 0,C 180,E1 -2805.314,E2 -2805.314} C_VEL
LIN {X 0,Y 558.82,Z 308.431,A -85,B 0,C 180,E1 -2808.325,E2 -2808.325} C_VEL
LIN {X 0,Y 558.863,Z 304.459,A -85,B 0,C 180,E1 -2810.617,E2 -2810.617} C_VEL
LIN {X 0,Y 558.929,Z 299.511,A -85,B 0,C 180,E1 -2813.378,E2 -2813.378} C_VEL
LIN {X 0,Y 558.924,Z 294.63,A -85,B 0,C 180,E1 -2816.11,E2 -2816.11} C_VEL
LIN {X 0,Y 558.935,Z 290.312,A -85,B 0,C 180,E1 -2818.543,E2 -2818.543} C_VEL
LIN {X 0,Y 558.99,Z 285.524,A -85,B 0,C 180,E1 -2821.246,E2 -2821.246} C_VEL
LIN {X 0,Y 559.052,Z 280.027,A -85,B 0,C 180,E1 -2824.159,E2 -2824.159} C_VEL
LIN {X 0,Y 559.133,Z 279.838,A -85,B 0,C 180,E1 -2826.443,E2 -2826.443} C_VEL
LIN {X 0,Y 559.18,Z 279.832,A -85,B 0,C 180,E1 -2828.934,E2 -2828.934} C_VEL
LIN {X 0,Y 559.165,Z 279.833,A -85,B 0,C 180,E1 -2831.77,E2 -2831.77} C_VEL
LIN {X 0,Y 559.135,Z 279.839,A -85,B 0,C 180,E1 -2834.74,E2 -2834.74} C_VEL
LIN {X 0,Y 559.161,Z 279.835,A -85,B 0,C 180,E1 -2837.256,E2 -2837.256} C_VEL
LIN {X 0,Y 559.187,Z 279.834,A -85,B 0,C 180,E1 -2840.135,E2 -2840.135} C_VEL
LIN {X 0,Y 559.134,Z 279.84,A -85,B 0,C 180,E1 -2842.891,E2 -2842.891} C_VEL
LIN {X 0,Y 559.095,Z 279.845,A -85,B 0,C 180,E1 -2845.551,E2 -2845.551} C_VEL
LIN {X 0,Y 559.047,Z 280.088,A -85,B 0,C 180,E1 -2846.069,E2 -2846.069} C_VEL
LIN {X 0,Y 558.975,Z 285.459,A -85,B 0,C 180,E1 -2848.969,E2 -2848.969} C_VEL
LIN {X 0,Y 558.944,Z 290.419,A -85,B 0,C 180,E1 -2851.662,E2 -2851.662} C_VEL
LIN {X 0,Y 558.973,Z 296.229,A -85,B 0,C 180,E1 -2854.859,E2 -2854.859} C_VEL
LIN {X 0,Y 558.893,Z 301.478,A -85,B 0,C 180,E1 -2857.837,E2 -2857.837} C_VEL
LIN {X 0,Y 558.875,Z 306.9,A -85,B 0,C 180,E1 -2860.916,E2 -2860.916} C_VEL
LIN {X 0,Y 558.791,Z 312.397,A -85,B 0,C 180,E1 -2863.937,E2 -2863.937} C_VEL
LIN {X 0,Y 558.808,Z 316.545,A -85,B 0,C 180,E1 -2866.175,E2 -2866.175} C_VEL
LIN {X 0,Y 558.823,Z 318.721,A -85,B 0,C 180,E1 -2867.263,E2 -2867.263} C_VEL
LIN {X 0,Y 559.982,Z 326.241,A -85,B 0,C 180,E1 -2867.451,E2 -2867.451} C_VEL
LIN {X 0,Y 559.874,Z 337.112,A -85,B 0,C 180,E1 -2867.77,E2 -2867.77} C_VEL
LIN {X 0,Y 559.701,Z 349.642,A -85,B 0,C 180,E1 -2868.277,E2 -2868.277} C_VEL
LIN {X 0,Y 559.566,Z 361.234,A -85,B 0,C 180,E1 -2868.91,E2 -2868.91} C_VEL
LIN {X 0,Y 559.427,Z 371.26,A -85,B 0,C 180,E1 -2869.596,E2 -2869.596} C_VEL
LIN {X 0,Y 559.299,Z 379.066,A -85,B 0,C 180,E1 -2870.233,E2 -2870.233} C_VEL
LIN {X 0,Y 559.197,Z 386.633,A -85,B 0,C 180,E1 -2870.961,E2 -2870.961} C_VEL
LIN {X 0,Y 559.051,Z 394.531,A -85,B 0,C 180,E1 -2871.869,E2 -2871.869} C_VEL
LIN {X 0,Y 558.985,Z 401.106,A -85,B 0,C 180,E1 -2872.777,E2 -2872.777} C_VEL
LIN {X 0,Y 558.913,Z 407.569,A -85,B 0,C 180,E1 -2873.864,E2 -2873.864} C_VEL
LIN {X 0,Y 558.798,Z 412.724,A -85,B 0,C 180,E1 -2874.949,E2 -2874.949} C_VEL
LIN {X 0,Y 558.844,Z 416.726,A -85,B 0,C 180,E1 -2876.034,E2 -2876.034} C_VEL
LIN {X 0,Y 558.799,Z 419.687,A -85,B 0,C 180,E1 -2877.116,E2 -2877.116} C_VEL
LIN {X 0,Y 558.745,Z 422.137,A -85,B 0,C 180,E1 -2878.558,E2 -2878.558} C_VEL
LIN {X 0,Y 558.741,Z 422.76,A -85,B 0,C 180,E1 -2879.279,E2 -2879.279} C_VEL
LIN {X 0,Y 558.741,Z 422.801,A -85,B 0,C 180,E1 -2880.721,E2 -2880.721} C_VEL
LIN {X 0,Y 558.746,Z 422.246,A -85,B 0,C 180,E1 -2881.441,E2 -2881.441} C_VEL
LIN {X 0,Y 558.8,Z 419.881,A -85,B 0,C 180,E1 -2882.884,E2 -2882.884} C_VEL
LIN {X 0,Y 558.844,Z 417.004,A -85,B 0,C 180,E1 -2883.966,E2 -2883.966} C_VEL
LIN {X 0,Y 558.798,Z 413.093,A -85,B 0,C 180,E1 -2885.051,E2 -2885.051} C_VEL
LIN {X 0,Y 558.914,Z 408.04,A -85,B 0,C 180,E1 -2886.136,E2 -2886.136} C_VEL
LIN {X 0,Y 558.975,Z 401.698,A -85,B 0,C 180,E1 -2887.223,E2 -2887.223} C_VEL
LIN {X 0,Y 559.073,Z 393.85,A -85,B 0,C 180,E1 -2888.312,E2 -2888.312} C_VEL
LIN {X 0,Y 559.223,Z 383.955,A -85,B 0,C 180,E1 -2889.403,E2 -2889.403} C_VEL
LIN {X 0,Y 559.393,Z 374.741,A -85,B 0,C 180,E1 -2890.222,E2 -2890.222} C_VEL
LIN {X 0,Y 559.461,Z 365.029,A -85,B 0,C 180,E1 -2890.936,E2 -2890.936} C_VEL
LIN {X 0,Y 559.597,Z 355.644,A -85,B 0,C 180,E1 -2891.501,E2 -2891.501} C_VEL
LIN {X 0,Y 559.737,Z 345.321,A -85,B 0,C 180,E1 -2892.003,E2 -2892.003} C_VEL
LIN {X 0,Y 559.94,Z 333.015,A -85,B 0,C 180,E1 -2892.458,E2 -2892.458} C_VEL
LIN {X 0,Y 559.786,Z 324.374,A -85,B 0,C 180,E1 -2892.692,E2 -2892.692} C_VEL
LIN {X 0,Y 558.788,Z 318.571,A -85,B 0,C 180,E1 -2892.83,E2 -2892.83} C_VEL
LIN {X 0,Y 558.827,Z 313.946,A -85,B 0,C 180,E1 -2895.314,E2 -2895.314} C_VEL
LIN {X 0,Y 558.819,Z 308.422,A -85,B 0,C 180,E1 -2898.325,E2 -2898.325} C_VEL
LIN {X 0,Y 558.86,Z 304.431,A -85,B 0,C 180,E1 -2900.617,E2 -2900.617} C_VEL
LIN {X 0,Y 558.926,Z 300.3,A -85,B 0,C 180,E1 -2902.942,E2 -2902.942} C_VEL
LIN {X 0,Y 558.913,Z 294.235,A -85,B 0,C 180,E1 -2906.111,E2 -2906.111} C_VEL
LIN {X 0,Y 558.859,Z 289.237,A -85,B 0,C 180,E1 -2908.547,E2 -2908.547} C_VEL
LIN {X 0,Y 558.823,Z 283.132,A -85,B 0,C 180,E1 -2911.218,E2 -2911.218} C_VEL
LIN {X 0,Y 558.837,Z 279.878,A -85,B 0,C 180,E1 -2912.584,E2 -2912.584} C_VEL
LIN {X 0,Y 559.114,Z 279.84,A -85,B 0,C 180,E1 -2914.447,E2 -2914.447} C_VEL
LIN {X 0,Y 559.141,Z 279.837,A -85,B 0,C 180,E1 -2917.109,E2 -2917.109} C_VEL
LIN {X 0,Y 559.162,Z 279.834,A -85,B 0,C 180,E1 -2919.941,E2 -2919.941} C_VEL
LIN {X 0,Y 559.152,Z 279.836,A -85,B 0,C 180,E1 -2922.744,E2 -2922.744} C_VEL
LIN {X 0,Y 559.155,Z 279.837,A -85,B 0,C 180,E1 -2925.761,E2 -2925.761} C_VEL
LIN {X 0,Y 559.159,Z 279.837,A -85,B 0,C 180,E1 -2928.229,E2 -2928.229} C_VEL
LIN {X 0,Y 559.175,Z 279.835,A -85,B 0,C 180,E1 -2931.192,E2 -2931.192} C_VEL
LIN {X 0,Y 559.166,Z 279.853,A -85,B 0,C 180,E1 -2932.421,E2 -2932.421} C_VEL
LIN {X 0,Y 560.276,Z 286.133,A -85,B 0,C 180,E1 -2934.296,E2 -2934.296} C_VEL
LIN {X 0,Y 560.061,Z 295.429,A -85,B 0,C 180,E1 -2936.902,E2 -2936.902} C_VEL
LIN {X 0,Y 559.906,Z 304.689,A -85,B 0,C 180,E1 -2939.445,E2 -2939.445} C_VEL
LIN {X 0,Y 559.732,Z 315.432,A -85,B 0,C 180,E1 -2942.317,E2 -2942.317} C_VEL
LIN {X 0,Y 559.532,Z 326.198,A -85,B 0,C 180,E1 -2945.122,E2 -2945.122} C_VEL
LIN {X 0,Y 559.415,Z 335.384,A -85,B 0,C 180,E1 -2947.469,E2 -2947.469} C_VEL
LIN {X 0,Y 559.281,Z 347.342,A -85,B 0,C 180,E1 -2950.469,E2 -2950.469} C_VEL
LIN {X 0,Y 559.174,Z 358.405,A -85,B 0,C 180,E1 -2953.197,E2 -2953.197} C_VEL
LIN {X 0,Y 559.033,Z 370.683,A -85,B 0,C 180,E1 -2956.181,E2 -2956.181} C_VEL
LIN {X 0,Y 559.004,Z 374.712,A -85,B 0,C 180,E1 -2957.151,E2 -2957.151} C_VEL
LIN {X 0,Y 560.041,Z 382.367,A -85,B 0,C 180,E1 -2957.314,E2 -2957.314} C_VEL
LIN {X 0,Y 559.911,Z 394.495,A -85,B 0,C 180,E1 -2957.633,E2 -2957.633} C_VEL
LIN {X 0,Y 559.736,Z 406.318,A -85,B 0,C 180,E1 -2958.08,E2 -2958.08} C_VEL
LIN {X 0,Y 559.57,Z 418.653,A -85,B 0,C 180,E1 -2958.708,E2 -2958.708} C_VEL
LIN {X 0,Y 559.424,Z 429.478,A -85,B 0,C 180,E1 -2959.413,E2 -2959.413} C_VEL
LIN {X 0,Y 559.298,Z 439.646,A -85,B 0,C 180,E1 -2960.233,E2 -2960.233} C_VEL
LIN {X 0,Y 559.134,Z 448.786,A -85,B 0,C 180,E1 -2961.143,E2 -2961.143} C_VEL
LIN {X 0,Y 559.009,Z 457.69,A -85,B 0,C 180,E1 -2962.233,E2 -2962.233} C_VEL
LIN {X 0,Y 558.925,Z 463.742,A -85,B 0,C 180,E1 -2963.14,E2 -2963.14} C_VEL
LIN {X 0,Y 558.936,Z 469.68,A -85,B 0,C 180,E1 -2964.227,E2 -2964.227} C_VEL
LIN {X 0,Y 558.826,Z 474.371,A -85,B 0,C 180,E1 -2965.311,E2 -2965.311} C_VEL
LIN {X 0,Y 558.836,Z 477.956,A -85,B 0,C 180,E1 -2966.395,E2 -2966.395} C_VEL
LIN {X 0,Y 558.799,Z 479.808,A -85,B 0,C 180,E1 -2967.116,E2 -2967.116} C_VEL
LIN {X 0,Y 558.747,Z 481.2,A -85,B 0,C 180,E1 -2967.837,E2 -2967.837} C_VEL
LIN {X 0,Y 558.741,Z 482.784,A -85,B 0,C 180,E1 -2969.279,E2 -2969.279} C_VEL
LIN {X 0,Y 558.74,Z 483,A -85,B 0,C 180,E1 -2970,E2 -2970} C_VEL
LIN {X 0,Y 558.745,Z 482.186,A -85,B 0,C 180,E1 -2971.442,E2 -2971.442} C_VEL
LIN {X 0,Y 558.747,Z 481.2,A -85,B 0,C 180,E1 -2972.163,E2 -2972.163} C_VEL
LIN {X 0,Y 558.799,Z 479.81,A -85,B 0,C 180,E1 -2972.884,E2 -2972.884} C_VEL
LIN {X 0,Y 558.844,Z 476.896,A -85,B 0,C 180,E1 -2973.966,E2 -2973.966} C_VEL
LIN {X 0,Y 558.798,Z 472.949,A -85,B 0,C 180,E1 -2975.051,E2 -2975.051} C_VEL
LIN {X 0,Y 558.922,Z 467.866,A -85,B 0,C 180,E1 -2976.136,E2 -2976.136} C_VEL
LIN {X 0,Y 558.977,Z 461.469,A -85,B 0,C 180,E1 -2977.223,E2 -2977.223} C_VEL
LIN {X 0,Y 559.099,Z 453.478,A -85,B 0,C 180,E1 -2978.312,E2 -2978.312} C_VEL
LIN {X 0,Y 559.195,Z 445.336,A -85,B 0,C 180,E1 -2979.221,E2 -2979.221} C_VEL
LIN {X 0,Y 559.358,Z 435.401,A -85,B 0,C 180,E1 -2980.131,E2 -2980.131} C_VEL
LIN {X 0,Y 559.504,Z 424.437,A -85,B 0,C 180,E1 -2980.935,E2 -2980.935} C_VEL
LIN {X 0,Y 559.636,Z 412.822,A -85,B 0,C 180,E1 -2981.61,E2 -2981.61} C_VEL
LIN {X 0,Y 559.779,Z 400.986,A -85,B 0,C 180,E1 -2982.14,E2 -2982.14} C_VEL
LIN {X 0,Y 559.963,Z 388.175,A -85,B 0,C 180,E1 -2982.55,E2 -2982.55} C_VEL
LIN {X 0,Y 559.835,Z 380.084,A -85,B 0,C 180,E1 -2982.737,E2 -2982.737} C_VEL
LIN {X 0,Y 559.004,Z 374.712,A -85,B 0,C 180,E1 -2982.849,E2 -2982.849} C_VEL
LIN {X 0,Y 559.088,Z 363.009,A -85,B 0,C 180,E1 -2985.68,E2 -2985.68} C_VEL
LIN {X 0,Y 559.189,Z 352.266,A -85,B 0,C 180,E1 -2988.313,E2 -2988.313} C_VEL
LIN {X 0,Y 559.341,Z 341.523,A -85,B 0,C 180,E1 -2990.983,E2 -2990.983} C_VEL
LIN {X 0,Y 559.527,Z 329.245,A -85,B 0,C 180,E1 -2994.093,E2 -2994.093} C_VEL
LIN {X 0,Y 559.653,Z 318.323,A -85,B 0,C 180,E1 -2996.924,E2 -2996.924} C_VEL
LIN {X 0,Y 559.879,Z 308.044,A -85,B 0,C 180,E1 -2999.648,E2 -2999.648} C_VEL
LIN {X 0,Y 560.04,Z 298.55,A -85,B 0,C 180,E1 -3002.231,E2 -3002.231} C_VEL
LIN {X 0,Y 560.22,Z 289.341,A -85,B 0,C 180,E1 -3004.806,E2 -3004.806} C_VEL
LIN {X 0,Y 560.008,Z 284.393,A -85,B 0,C 180,E1 -3006.146,E2 -3006.146} C_VEL
LIN {X 0,Y 559.144,Z 279.839,A -85,B 0,C 180,E1 -3007.499,E2 -3007.499} C_VEL
LIN {X 0,Y 559.157,Z 279.832,A -85,B 0,C 180,E1 -3009.941,E2 -3009.941} C_VEL
LIN {X 0,Y 559.143,Z 279.84,A -85,B 0,C 180,E1 -3012.745,E2 -3012.745} C_VEL
LIN {X 0,Y 559.149,Z 279.833,A -85,B 0,C 180,E1 -3015.761,E2 -3015.761} C_VEL
LIN {X 0,Y 559.158,Z 279.837,A -85,B 0,C 180,E1 -3018.229,E2 -3018.229} C_VEL
LIN {X 0,Y 559.179,Z 279.828,A -85,B 0,C 180,E1 -3021.192,E2 -3021.192} C_VEL
LIN {X 0,Y 559.142,Z 279.838,A -85,B 0,C 180,E1 -3023.789,E2 -3023.789} C_VEL
LIN {X 0,Y 559.166,Z 279.832,A -85,B 0,C 180,E1 -3026.425,E2 -3026.425} C_VEL
LIN {X 0,Y 559.158,Z 279.831,A -85,B 0,C 180,E1 -3028.981,E2 -3028.981} C_VEL
LIN {X 0,Y 559.172,Z 279.837,A -85,B 0,C 180,E1 -3031.619,E2 -3031.619} C_VEL
LIN {X 0,Y 559.176,Z 279.832,A -85,B 0,C 180,E1 -3033.903,E2 -3033.903} C_VEL
LIN {X 0,Y 559.016,Z 279.855,A -85,B 0,C 180,E1 -3036.602,E2 -3036.602} C_VEL
LIN {X 0,Y 558.869,Z 280.3,A -85,B 0,C 180,E1 -3037.836,E2 -3037.836} C_VEL
LIN {X 0,Y 558.843,Z 282.313,A -85,B 0,C 180,E1 -3040.15,E2 -3040.15} C_VEL
LIN {X 0,Y 558.783,Z 285.088,A -85,B 0,C 180,E1 -3043.185,E2 -3043.185} C_VEL
LIN {X 0,Y 558.771,Z 288.604,A -85,B 0,C 180,E1 -3046.174,E2 -3046.174} C_VEL
LIN {X 0,Y 558.771,Z 289.895,A -85,B 0,C 180,E1 -3047.262,E2 -3047.262} C_VEL
LIN {X 0,Y 559.965,Z 298.291,A -85,B 0,C 180,E1 -3047.496,E2 -3047.496} C_VEL
LIN {X 0,Y 559.776,Z 311.431,A -85,B 0,C 180,E1 -3047.929,E2 -3047.929} C_VEL
LIN {X 0,Y 559.62,Z 322.192,A -85,B 0,C 180,E1 -3048.408,E2 -3048.408} C_VEL
LIN {X 0,Y 559.528,Z 331.306,A -85,B 0,C 180,E1 -3048.917,E2 -3048.917} C_VEL
LIN {X 0,Y 559.456,Z 340.029,A -85,B 0,C 180,E1 -3049.505,E2 -3049.505} C_VEL
LIN {X 0,Y 559.3,Z 349.046,A -85,B 0,C 180,E1 -3050.233,E2 -3050.233} C_VEL
LIN {X 0,Y 559.166,Z 356.605,A -85,B 0,C 180,E1 -3050.961,E2 -3050.961} C_VEL
LIN {X 0,Y 559.05,Z 364.543,A -85,B 0,C 180,E1 -3051.87,E2 -3051.87} C_VEL
LIN {X 0,Y 558.967,Z 372.469,A -85,B 0,C 180,E1 -3052.977,E2 -3052.977} C_VEL
LIN {X 0,Y 558.936,Z 379.425,A -85,B 0,C 180,E1 -3054.227,E2 -3054.227} C_VEL
LIN {X 0,Y 558.826,Z 384.153,A -85,B 0,C 180,E1 -3055.311,E2 -3055.311} C_VEL
LIN {X 0,Y 558.836,Z 387.783,A -85,B 0,C 180,E1 -3056.395,E2 -3056.395} C_VEL
LIN {X 0,Y 558.799,Z 389.678,A -85,B 0,C 180,E1 -3057.116,E2 -3057.116} C_VEL
LIN {X 0,Y 558.747,Z 391.136,A -85,B 0,C 180,E1 -3057.837,E2 -3057.837} C_VEL
LIN {X 0,Y 558.741,Z 392.74,A -85,B 0,C 180,E1 -3059.279,E2 -3059.279} C_VEL
LIN {X 0,Y 558.74,Z 392.996,A -85,B 0,C 180,E1 -3060,E2 -3060} C_VEL
LIN {X 0,Y 558.746,Z 392.214,A -85,B 0,C 180,E1 -3061.442,E2 -3061.442} C_VEL
LIN {X 0,Y 558.747,Z 391.28,A -85,B 0,C 180,E1 -3062.163,E2 -3062.163} C_VEL
LIN {X 0,Y 558.836,Z 388.043,A -85,B 0,C 180,E1 -3063.605,E2 -3063.605} C_VEL
LIN {X 0,Y 558.826,Z 384.495,A -85,B 0,C 180,E1 -3064.689,E2 -3064.689} C_VEL
LIN {X 0,Y 558.928,Z 379.85,A -85,B 0,C 180,E1 -3065.773,E2 -3065.773} C_VEL
LIN {X 0,Y 558.939,Z 372.908,A -85,B 0,C 180,E1 -3067.042,E2 -3067.042} C_VEL
LIN {X 0,Y 559.04,Z 365.295,A -85,B 0,C 180,E1 -3068.131,E2 -3068.131} C_VEL
LIN {X 0,Y 559.172,Z 357.487,A -85,B 0,C 180,E1 -3069.039,E2 -3069.039} C_VEL
LIN {X 0,Y 559.292,Z 349.035,A -85,B 0,C 180,E1 -3069.858,E2 -3069.858} C_VEL
LIN {X 0,Y 559.415,Z 340.004,A -85,B 0,C 180,E1 -3070.588,E2 -3070.588} C_VEL
LIN {X 0,Y 559.53,Z 330.545,A -85,B 0,C 180,E1 -3071.219,E2 -3071.219} C_VEL
LIN {X 0,Y 559.689,Z 320.32,A -85,B 0,C 180,E1 -3071.774,E2 -3071.774} C_VEL
LIN {X 0,Y 559.859,Z 308.463,A -85,B 0,C 180,E1 -3072.276,E2 -3072.276} C_VEL
LIN {X 0,Y 559.816,Z 296.399,A -85,B 0,C 180,E1 -3072.645,E2 -3072.645} C_VEL
LIN {X 0,Y 558.749,Z 289.892,A -85,B 0,C 180,E1 -3072.831,E2 -3072.831} C_VEL
LIN {X 0,Y 558.728,Z 286.952,A -85,B 0,C 180,E1 -3075.317,E2 -3075.317} C_VEL
LIN {X 0,Y 558.745,Z 284.326,A -85,B 0,C 180,E1 -3077.57,E2 -3077.57} C_VEL
LIN {X 0,Y 558.783,Z 281.897,A -85,B 0,C 180,E1 -3079.852,E2 -3079.852} C_VEL
LIN {X 0,Y 558.808,Z 280.239,A -85,B 0,C 180,E1 -3081.458,E2 -3081.458} C_VEL
LIN {X 0,Y 558.92,Z 279.866,A -85,B 0,C 180,E1 -3082.942,E2 -3082.942} C_VEL
LIN {X 0,Y 559.132,Z 279.833,A -85,B 0,C 180,E1 -3085.3,E2 -3085.3} C_VEL
LIN {X 0,Y 559.164,Z 279.832,A -85,B 0,C 180,E1 -3086.704,E2 -3086.704} C_VEL
LIN {X 0,Y 558.515,Z 279.917,A -85,B 0,C 180,E1 -3087.305,E2 -3087.305} C_VEL
LIN {X 0,Y 555.653,Z 280.271,A -85,B 0,C 180,E1 -3088.281,E2 -3088.281} C_VEL
LIN {X 0,Y 553.226,Z 280.57,A -85,B 0,C 180,E1 -3089.067,E2 -3089.067} C_VEL
LIN {X 0,Y 552.191,Z 280.697,A -85,B 0,C 180,E1 -3089.673,E2 -3089.673} C_VEL
LIN {X 0,Y 552.112,Z 280.708,A -85,B 0,C 180,E1 -3089.879,E2 -3089.879} C_VEL
LIN {X 0,Y 552.116,Z 280.709,A -85,B 0,C 180,E1 -3092.846,E2 -3092.846} C_VEL
LIN {X 0,Y 552.079,Z 280.71,A -85,B 0,C 180,E1 -3095.44,E2 -3095.44} C_VEL
LIN {X 0,Y 552.101,Z 280.713,A -85,B 0,C 180,E1 -3097.886,E2 -3097.886} C_VEL
LIN {X 0,Y 552.113,Z 280.711,A -85,B 0,C 180,E1 -3100.481,E2 -3100.481} C_VEL
LIN {X 0,Y 552.123,Z 280.709,A -85,B 0,C 180,E1 -3103.485,E2 -3103.485} C_VEL
LIN {X 0,Y 552.11,Z 280.708,A -85,B 0,C 180,E1 -3106.576,E2 -3106.576} C_VEL
LIN {X 0,Y 552.112,Z 280.713,A -85,B 0,C 180,E1 -3109.519,E2 -3109.519} C_VEL
LIN {X 0,Y 552.096,Z 280.71,A -85,B 0,C 180,E1 -3112.336,E2 -3112.336} C_VEL
LIN {X 0,Y 552.061,Z 280.717,A -85,B 0,C 180,E1 -3115.049,E2 -3115.049} C_VEL
LIN {X 0,Y 552.005,Z 280.745,A -85,B 0,C 180,E1 -3115.93,E2 -3115.93} C_VEL
LIN {X 0,Y 551.927,Z 285.717,A -85,B 0,C 180,E1 -3118.556,E2 -3118.556} C_VEL
LIN {X 0,Y 551.868,Z 290.897,A -85,B 0,C 180,E1 -3121.488,E2 -3121.488} C_VEL
LIN {X 0,Y 551.884,Z 295.906,A -85,B 0,C 180,E1 -3124.343,E2 -3124.343} C_VEL
LIN {X 0,Y 551.847,Z 300.175,A -85,B 0,C 180,E1 -3126.747,E2 -3126.747} C_VEL
LIN {X 0,Y 551.792,Z 304.374,A -85,B 0,C 180,E1 -3129.107,E2 -3129.107} C_VEL
LIN {X 0,Y 551.757,Z 308.462,A -85,B 0,C 180,E1 -3131.431,E2 -3131.431} C_VEL
LIN {X 0,Y 551.723,Z 312.444,A -85,B 0,C 180,E1 -3133.725,E2 -3133.725} C_VEL
LIN {X 0,Y 551.726,Z 316.546,A -85,B 0,C 180,E1 -3135.994,E2 -3135.994} C_VEL
LIN {X 0,Y 551.71,Z 318.625,A -85,B 0,C 180,E1 -3137.096,E2 -3137.096} C_VEL
LIN {X 0,Y 553.022,Z 327.131,A -85,B 0,C 180,E1 -3137.313,E2 -3137.313} C_VEL
LIN {X 0,Y 552.915,Z 337.066,A -85,B 0,C 180,E1 -3137.614,E2 -3137.614} C_VEL
LIN {X 0,Y 552.764,Z 347.403,A -85,B 0,C 180,E1 -3138.03,E2 -3138.03} C_VEL
LIN {X 0,Y 552.632,Z 356.287,A -85,B 0,C 180,E1 -3138.479,E2 -3138.479} C_VEL
LIN {X 0,Y 552.504,Z 364.809,A -85,B 0,C 180,E1 -3139,E2 -3139} C_VEL
LIN {X 0,Y 552.386,Z 373.615,A -85,B 0,C 180,E1 -3139.647,E2 -3139.647} C_VEL
LIN {X 0,Y 552.246,Z 381.068,A -85,B 0,C 180,E1 -3140.292,E2 -3140.292} C_VEL
LIN {X 0,Y 552.124,Z 388.329,A -85,B 0,C 180,E1 -3141.029,E2 -3141.029} C_VEL
LIN {X 0,Y 551.985,Z 395.936,A -85,B 0,C 180,E1 -3141.949,E2 -3141.949} C_VEL
LIN {X 0,Y 551.895,Z 402.394,A -85,B 0,C 180,E1 -3142.886,E2 -3142.886} C_VEL
LIN {X 0,Y 551.839,Z 408.163,A -85,B 0,C 180,E1 -3143.901,E2 -3143.901} C_VEL
LIN {X 0,Y 551.723,Z 412.702,A -85,B 0,C 180,E1 -3144.884,E2 -3144.884} C_VEL
LIN {X 0,Y 551.764,Z 416.7,A -85,B 0,C 180,E1 -3145.983,E2 -3145.983} C_VEL
LIN {X 0,Y 551.723,Z 419.661,A -85,B 0,C 180,E1 -3147.079,E2 -3147.079} C_VEL
LIN {X 0,Y 551.645,Z 422.148,A -85,B 0,C 180,E1 -3148.54,E2 -3148.54} C_VEL
LIN {X 0,Y 551.642,Z 422.748,A -85,B 0,C 180,E1 -3149.27,E2 -3149.27} C_VEL
LIN {X 0,Y 551.641,Z 422.809,A -85,B 0,C 180,E1 -3150.73,E2 -3150.73} C_VEL
LIN {X 0,Y 551.646,Z 422.236,A -85,B 0,C 180,E1 -3151.46,E2 -3151.46} C_VEL
LIN {X 0,Y 551.724,Z 419.88,A -85,B 0,C 180,E1 -3152.921,E2 -3152.921} C_VEL
LIN {X 0,Y 551.764,Z 416.997,A -85,B 0,C 180,E1 -3154.017,E2 -3154.017} C_VEL
LIN {X 0,Y 551.723,Z 413.082,A -85,B 0,C 180,E1 -3155.116,E2 -3155.116} C_VEL
LIN {X 0,Y 551.837,Z 408.632,A -85,B 0,C 180,E1 -3156.098,E2 -3156.098} C_VEL
LIN {X 0,Y 551.887,Z 402.842,A -85,B 0,C 180,E1 -3157.132,E2 -3157.132} C_VEL
LIN {X 0,Y 551.983,Z 396.605,A -85,B 0,C 180,E1 -3158.051,E2 -3158.051} C_VEL
LIN {X 0,Y 552.102,Z 389.119,A -85,B 0,C 180,E1 -3158.971,E2 -3158.971} C_VEL
LIN {X 0,Y 552.225,Z 381.999,A -85,B 0,C 180,E1 -3159.708,E2 -3159.708} C_VEL
LIN {X 0,Y 552.404,Z 373.583,A -85,B 0,C 180,E1 -3160.445,E2 -3160.445} C_VEL
LIN {X 0,Y 552.523,Z 364.118,A -85,B 0,C 180,E1 -3161.137,E2 -3161.137} C_VEL
LIN {X 0,Y 552.698,Z 352.301,A -85,B 0,C 180,E1 -3161.832,E2 -3161.832} C_VEL
LIN {X 0,Y 552.857,Z 340.836,A -85,B 0,C 180,E1 -3162.341,E2 -3162.341} C_VEL
LIN {X 0,Y 552.997,Z 329.629,A -85,B 0,C 180,E1 -3162.71,E2 -3162.71} C_VEL
LIN {X 0,Y 552.755,Z 324.821,A -85,B 0,C 180,E1 -3162.845,E2 -3162.845} C_VEL
LIN {X 0,Y 551.698,Z 318.57,A -85,B 0,C 180,E1 -3162.998,E2 -3162.998} C_VEL
LIN {X 0,Y 551.739,Z 313.945,A -85,B 0,C 180,E1 -3165.515,E2 -3165.515} C_VEL
LIN {X 0,Y 551.744,Z 309.986,A -85,B 0,C 180,E1 -3167.801,E2 -3167.801} C_VEL
LIN {X 0,Y 551.79,Z 305.938,A -85,B 0,C 180,E1 -3170.114,E2 -3170.114} C_VEL
LIN {X 0,Y 551.836,Z 301.755,A -85,B 0,C 180,E1 -3172.462,E2 -3172.462} C_VEL
LIN {X 0,Y 551.905,Z 296.709,A -85,B 0,C 180,E1 -3175.294,E2 -3175.294} C_VEL
LIN {X 0,Y 551.87,Z 291.06,A -85,B 0,C 180,E1 -3178.513,E2 -3178.513} C_VEL
LIN {X 0,Y 551.909,Z 287.365,A -85,B 0,C 180,E1 -3180.621,E2 -3180.621} C_VEL
LIN {X 0,Y 551.941,Z 282.626,A -85,B 0,C 180,E1 -3183.198,E2 -3183.198} C_VEL
LIN {X 0,Y 551.987,Z 280.732,A -85,B 0,C 180,E1 -3184.195,E2 -3184.195} C_VEL
LIN {X 0,Y 552.102,Z 280.714,A -85,B 0,C 180,E1 -3186.748,E2 -3186.748} C_VEL
LIN {X 0,Y 552.136,Z 280.711,A -85,B 0,C 180,E1 -3189.527,E2 -3189.527} C_VEL
LIN {X 0,Y 552.133,Z 280.714,A -85,B 0,C 180,E1 -3192.425,E2 -3192.425} C_VEL
LIN {X 0,Y 552.095,Z 280.714,A -85,B 0,C 180,E1 -3195.562,E2 -3195.562} C_VEL
LIN {X 0,Y 552.123,Z 280.711,A -85,B 0,C 180,E1 -3198.554,E2 -3198.554} C_VEL
LIN {X 0,Y 552.121,Z 280.714,A -85,B 0,C 180,E1 -3201.411,E2 -3201.411} C_VEL
LIN {X 0,Y 552.076,Z 280.719,A -85,B 0,C 180,E1 -3204.155,E2 -3204.155} C_VEL
LIN {X 0,Y 552.01,Z 280.751,A -85,B 0,C 180,E1 -3206.041,E2 -3206.041} C_VEL
LIN {X 0,Y 551.901,Z 286.917,A -85,B 0,C 180,E1 -3209.378,E2 -3209.378} C_VEL
LIN {X 0,Y 551.873,Z 291.473,A -85,B 0,C 180,E1 -3211.888,E2 -3211.888} C_VEL
LIN {X 0,Y 551.905,Z 296.566,A -85,B 0,C 180,E1 -3214.706,E2 -3214.706} C_VEL
LIN {X 0,Y 551.818,Z 301.559,A -85,B 0,C 180,E1 -3217.537,E2 -3217.537} C_VEL
LIN {X 0,Y 551.821,Z 307.071,A -85,B 0,C 180,E1 -3220.662,E2 -3220.662} C_VEL
LIN {X 0,Y 551.723,Z 312.46,A -85,B 0,C 180,E1 -3223.725,E2 -3223.725} C_VEL
LIN {X 0,Y 551.726,Z 316.546,A -85,B 0,C 180,E1 -3225.994,E2 -3225.994} C_VEL
LIN {X 0,Y 551.71,Z 318.71,A -85,B 0,C 180,E1 -3227.096,E2 -3227.096} C_VEL
LIN {X 0,Y 553.041,Z 327.153,A -85,B 0,C 180,E1 -3227.314,E2 -3227.314} C_VEL
LIN {X 0,Y 552.926,Z 338.46,A -85,B 0,C 180,E1 -3227.661,E2 -3227.661} C_VEL
LIN {X 0,Y 552.738,Z 350.494,A -85,B 0,C 180,E1 -3228.169,E2 -3228.169} C_VEL
LIN {X 0,Y 552.588,Z 361.52,A -85,B 0,C 180,E1 -3228.787,E2 -3228.787} C_VEL
LIN {X 0,Y 552.427,Z 371.255,A -85,B 0,C 180,E1 -3229.462,E2 -3229.462} C_VEL
LIN {X 0,Y 552.27,Z 379.06,A -85,B 0,C 180,E1 -3230.108,E2 -3230.108} C_VEL
LIN {X 0,Y 552.153,Z 386.627,A -85,B 0,C 180,E1 -3230.845,E2 -3230.845} C_VEL
LIN {X 0,Y 552.014,Z 394.525,A -85,B 0,C 180,E1 -3231.765,E2 -3231.765} C_VEL
LIN {X 0,Y 551.913,Z 401.1,A -85,B 0,C 180,E1 -3232.684,E2 -3232.684} C_VEL
LIN {X 0,Y 551.811,Z 406.837,A -85,B 0,C 180,E1 -3233.65,E2 -3233.65} C_VEL
LIN {X 0,Y 551.803,Z 411.122,A -85,B 0,C 180,E1 -3234.519,E2 -3234.519} C_VEL
LIN {X 0,Y 551.767,Z 415.474,A -85,B 0,C 180,E1 -3235.617,E2 -3235.617} C_VEL
LIN {X 0,Y 551.751,Z 417.836,A -85,B 0,C 180,E1 -3236.348,E2 -3236.348} C_VEL
LIN {X 0,Y 551.723,Z 419.687,A -85,B 0,C 180,E1 -3237.079,E2 -3237.079} C_VEL
LIN {X 0,Y 551.645,Z 422.136,A -85,B 0,C 180,E1 -3238.54,E2 -3238.54} C_VEL
LIN {X 0,Y 551.642,Z 422.761,A -85,B 0,C 180,E1 -3239.27,E2 -3239.27} C_VEL
LIN {X 0,Y 551.641,Z 422.799,A -85,B 0,C 180,E1 -3240.73,E2 -3240.73} C_VEL
LIN {X 0,Y 551.646,Z 422.245,A -85,B 0,C 180,E1 -3241.46,E2 -3241.46} C_VEL
LIN {X 0,Y 551.724,Z 419.874,A -85,B 0,C 180,E1 -3242.921,E2 -3242.921} C_VEL
LIN {X 0,Y 551.764,Z 416.995,A -85,B 0,C 180,E1 -3244.017,E2 -3244.017} C_VEL
LIN {X 0,Y 551.723,Z 413.082,A -85,B 0,C 180,E1 -3245.116,E2 -3245.116} C_VEL
LIN {X 0,Y 551.84,Z 408.633,A -85,B 0,C 180,E1 -3246.099,E2 -3246.099} C_VEL
LIN {X 0,Y 551.886,Z 402.846,A -85,B 0,C 180,E1 -3247.132,E2 -3247.132} C_VEL
LIN {X 0,Y 551.983,Z 396.61,A -85,B 0,C 180,E1 -3248.051,E2 -3248.051} C_VEL
LIN {X 0,Y 552.105,Z 389.114,A -85,B 0,C 180,E1 -3248.971,E2 -3248.971} C_VEL
LIN {X 0,Y 552.228,Z 381.995,A -85,B 0,C 180,E1 -3249.708,E2 -3249.708} C_VEL
LIN {X 0,Y 552.384,Z 373.568,A -85,B 0,C 180,E1 -3250.446,E2 -3250.446} C_VEL
LIN {X 0,Y 552.478,Z 365.091,A -85,B 0,C 180,E1 -3251.07,E2 -3251.07} C_VEL
LIN {X 0,Y 552.612,Z 355.844,A -85,B 0,C 180,E1 -3251.635,E2 -3251.635} C_VEL
LIN {X 0,Y 552.775,Z 346.328,A -85,B 0,C 180,E1 -3252.11,E2 -3252.11} C_VEL
LIN {X 0,Y 552.966,Z 335.662,A -85,B 0,C 180,E1 -3252.525,E2 -3252.525} C_VEL
LIN {X 0,Y 552.855,Z 325.226,A -85,B 0,C 180,E1 -3252.83,E2 -3252.83} C_VEL
LIN {X 0,Y 551.691,Z 318.57,A -85,B 0,C 180,E1 -3252.998,E2 -3252.998} C_VEL
LIN {X 0,Y 551.739,Z 313.945,A -85,B 0,C 180,E1 -3255.515,E2 -3255.515} C_VEL
LIN {X 0,Y 551.744,Z 310.025,A -85,B 0,C 180,E1 -3257.801,E2 -3257.801} C_VEL
LIN {X 0,Y 551.789,Z 305.919,A -85,B 0,C 180,E1 -3260.114,E2 -3260.114} C_VEL
LIN {X 0,Y 551.839,Z 301.776,A -85,B 0,C 180,E1 -3262.462,E2 -3262.462} C_VEL
LIN {X 0,Y 551.86,Z 296.392,A -85,B 0,C 180,E1 -3265.285,E2 -3265.285} C_VEL
LIN {X 0,Y 551.803,Z 292.462,A -85,B 0,C 180,E1 -3267.291,E2 -3267.291} C_VEL
LIN {X 0,Y 551.715,Z 286.518,A -85,B 0,C 180,E1 -3269.978,E2 -3269.978} C_VEL
LIN {X 0,Y 551.758,Z 280.76,A -85,B 0,C 180,E1 -3272.424,E2 -3272.424} C_VEL
LIN {X 0,Y 552.063,Z 280.72,A -85,B 0,C 180,E1 -3274.159,E2 -3274.159} C_VEL
LIN {X 0,Y 552.105,Z 280.714,A -85,B 0,C 180,E1 -3276.747,E2 -3276.747} C_VEL
LIN {X 0,Y 552.131,Z 280.71,A -85,B 0,C 180,E1 -3279.527,E2 -3279.527} C_VEL
LIN {X 0,Y 552.111,Z 280.712,A -85,B 0,C 180,E1 -3282.427,E2 -3282.427} C_VEL
LIN {X 0,Y 552.101,Z 280.716,A -85,B 0,C 180,E1 -3285.563,E2 -3285.563} C_VEL
LIN {X 0,Y 552.122,Z 280.712,A -85,B 0,C 180,E1 -3288.679,E2 -3288.679} C_VEL
LIN {X 0,Y 552.118,Z 280.713,A -85,B 0,C 180,E1 -3291.411,E2 -3291.411} C_VEL
LIN {X 0,Y 552.111,Z 280.83,A -85,B 0,C 180,E1 -3292.178,E2 -3292.178} C_VEL
LIN {X 0,Y 553.355,Z 287.668,A -85,B 0,C 180,E1 -3294.251,E2 -3294.251} C_VEL
LIN {X 0,Y 553.14,Z 297.392,A -85,B 0,C 180,E1 -3296.99,E2 -3296.99} C_VEL
LIN {X 0,Y 552.948,Z 307.529,A -85,B 0,C 180,E1 -3299.801,E2 -3299.801} C_VEL
LIN {X 0,Y 552.716,Z 318.502,A -85,B 0,C 180,E1 -3302.758,E2 -3302.758} C_VEL
LIN {X 0,Y 552.524,Z 329.245,A -85,B 0,C 180,E1 -3305.582,E2 -3305.582} C_VEL
LIN {X 0,Y 552.384,Z 339.988,A -85,B 0,C 180,E1 -3308.348,E2 -3308.348} C_VEL
LIN {X 0,Y 552.193,Z 352.266,A -85,B 0,C 180,E1 -3311.447,E2 -3311.447} C_VEL
LIN {X 0,Y 552.041,Z 363.009,A -85,B 0,C 180,E1 -3314.114,E2 -3314.114} C_VEL
LIN {X 0,Y 551.955,Z 374.712,A -85,B 0,C 180,E1 -3316.985,E2 -3316.985} C_VEL
LIN {X 0,Y 553.094,Z 383.507,A -85,B 0,C 180,E1 -3317.175,E2 -3317.175} C_VEL
LIN {X 0,Y 552.951,Z 395.875,A -85,B 0,C 180,E1 -3317.522,E2 -3317.522} C_VEL
LIN {X 0,Y 552.763,Z 407.509,A -85,B 0,C 180,E1 -3317.983,E2 -3317.983} C_VEL
LIN {X 0,Y 552.593,Z 419.257,A -85,B 0,C 180,E1 -3318.6,E2 -3318.6} C_VEL
LIN {X 0,Y 552.41,Z 430.746,A -85,B 0,C 180,E1 -3319.369,E2 -3319.369} C_VEL
LIN {X 0,Y 552.233,Z 441.6,A -85,B 0,C 180,E1 -3320.292,E2 -3320.292} C_VEL
LIN {X 0,Y 552.079,Z 450.412,A -85,B 0,C 180,E1 -3321.213,E2 -3321.213} C_VEL
LIN {X 0,Y 551.95,Z 459.001,A -85,B 0,C 180,E1 -3322.317,E2 -3322.317} C_VEL
LIN {X 0,Y 551.823,Z 465.868,A -85,B 0,C 180,E1 -3323.418,E2 -3323.418} C_VEL
LIN {X 0,Y 551.804,Z 471.366,A -85,B 0,C 180,E1 -3324.519,E2 -3324.519} C_VEL
LIN {X 0,Y 551.764,Z 475.677,A -85,B 0,C 180,E1 -3325.617,E2 -3325.617} C_VEL
LIN {X 0,Y 551.75,Z 477.957,A -85,B 0,C 180,E1 -3326.348,E2 -3326.348} C_VEL
LIN {X 0,Y 551.723,Z 479.808,A -85,B 0,C 180,E1 -3327.079,E2 -3327.079} C_VEL
LIN {X 0,Y 551.657,Z 481.199,A -85,B 0,C 180,E1 -3327.81,E2 -3327.81} C_VEL
LIN {X 0,Y 551.641,Z 482.785,A -85,B 0,C 180,E1 -3329.27,E2 -3329.27} C_VEL
LIN {X 0,Y 551.64,Z 483,A -85,B 0,C 180,E1 -3330,E2 -3330} C_VEL
LIN {X 0,Y 551.645,Z 482.186,A -85,B 0,C 180,E1 -3331.46,E2 -3331.46} C_VEL
LIN {X 0,Y 551.657,Z 481.2,A -85,B 0,C 180,E1 -3332.19,E2 -3332.19} C_VEL
LIN {X 0,Y 551.723,Z 479.81,A -85,B 0,C 180,E1 -3332.921,E2 -3332.921} C_VEL
LIN {X 0,Y 551.764,Z 476.896,A -85,B 0,C 180,E1 -3334.017,E2 -3334.017} C_VEL
LIN {X 0,Y 551.724,Z 472.949,A -85,B 0,C 180,E1 -3335.116,E2 -3335.116} C_VEL
LIN {X 0,Y 551.825,Z 467.189,A -85,B 0,C 180,E1 -3336.341,E2 -3336.341} C_VEL
LIN {X 0,Y 551.926,Z 460.237,A -85,B 0,C 180,E1 -3337.5,E2 -3337.5} C_VEL
LIN {X 0,Y 552.082,Z 451.99,A -85,B 0,C 180,E1 -3338.602,E2 -3338.602} C_VEL
LIN {X 0,Y 552.201,Z 443.538,A -85,B 0,C 180,E1 -3339.524,E2 -3339.524} C_VEL
LIN {X 0,Y 552.423,Z 433.096,A -85,B 0,C 180,E1 -3340.445,E2 -3340.445} C_VEL
LIN {X 0,Y 552.578,Z 421.349,A -85,B 0,C 180,E1 -3341.275,E2 -3341.275} C_VEL
LIN {X 0,Y 552.737,Z 409.483,A -85,B 0,C 180,E1 -3341.924,E2 -3341.924} C_VEL
LIN {X 0,Y 552.927,Z 397.171,A -85,B 0,C 180,E1 -3342.432,E2 -3342.432} C_VEL
LIN {X 0,Y 553.07,Z 384.518,A -85,B 0,C 180,E1 -3342.802,E2 -3342.802} C_VEL
LIN {X 0,Y 552.718,Z 379.514,A -85,B 0,C 180,E1 -3342.915,E2 -3342.915} C_VEL
LIN {X 0,Y 551.955,Z 374.712,A -85,B 0,C 180,E1 -3343.015,E2 -3343.015} C_VEL
LIN {X 0,Y 552.041,Z 363.009,A -85,B 0,C 180,E1 -3345.886,E2 -3345.886} C_VEL
LIN {X 0,Y 552.193,Z 352.266,A -85,B 0,C 180,E1 -3348.553,E2 -3348.553} C_VEL
LIN {X 0,Y 552.384,Z 339.988,A -85,B 0,C 180,E1 -3351.652,E2 -3351.652} C_VEL
LIN {X 0,Y 552.524,Z 329.245,A -85,B 0,C 180,E1 -3354.418,E2 -3354.418} C_VEL
LIN {X 0,Y 552.716,Z 318.502,A -85,B 0,C 180,E1 -3357.242,E2 -3357.242} C_VEL
LIN {X 0,Y 552.948,Z 307.529,A -85,B 0,C 180,E1 -3360.199,E2 -3360.199} C_VEL
LIN {X 0,Y 553.14,Z 297.392,A -85,B 0,C 180,E1 -3363.01,E2 -3363.01} C_VEL
LIN {X 0,Y 553.277,Z 289.229,A -85,B 0,C 180,E1 -3365.236,E2 -3365.236} C_VEL
LIN {X 0,Y 553.034,Z 285.639,A -85,B 0,C 180,E1 -3366.223,E2 -3366.223} C_VEL
LIN {X 0,Y 552.103,Z 280.715,A -85,B 0,C 180,E1 -3367.703,E2 -3367.703} C_VEL
LIN {X 0,Y 552.107,Z 280.715,A -85,B 0,C 180,E1 -3370.482,E2 -3370.482} C_VEL
LIN {X 0,Y 552.094,Z 280.712,A -85,B 0,C 180,E1 -3373.482,E2 -3373.482} C_VEL
LIN {X 0,Y 552.109,Z 280.716,A -85,B 0,C 180,E1 -3376.576,E2 -3376.576} C_VEL
LIN {X 0,Y 552.112,Z 280.709,A -85,B 0,C 180,E1 -3379.519,E2 -3379.519} C_VEL
LIN {X 0,Y 552.096,Z 280.717,A -85,B 0,C 180,E1 -3382.336,E2 -3382.336} C_VEL
LIN {X 0,Y 552.086,Z 280.712,A -85,B 0,C 180,E1 -3385.051,E2 -3385.051} C_VEL
LIN {X 0,Y 552.119,Z 280.714,A -85,B 0,C 180,E1 -3387.681,E2 -3387.681} C_VEL
LIN {X 0,Y 552.115,Z 280.71,A -85,B 0,C 180,E1 -3390.235,E2 -3390.235} C_VEL
LIN {X 0,Y 552.142,Z 280.708,A -85,B 0,C 180,E1 -3393,E2 -3393} C_VEL
LIN {X 0,Y 552.054,Z 280.722,A -85,B 0,C 180,E1 -3395.158,E2 -3395.158} C_VEL
LIN {X 0,Y 551.84,Z 280.882,A -85,B 0,C 180,E1 -3397.538,E2 -3397.538} C_VEL
LIN {X 0,Y 551.841,Z 283.104,A -85,B 0,C 180,E1 -3399.888,E2 -3399.888} C_VEL
LIN {X 0,Y 551.723,Z 285.689,A -85,B 0,C 180,E1 -3402.964,E2 -3402.964} C_VEL
LIN {X 0,Y 551.684,Z 288.605,A -85,B 0,C 180,E1 -3405.993,E2 -3405.993} C_VEL
LIN {X 0,Y 551.661,Z 289.896,A -85,B 0,C 180,E1 -3407.095,E2 -3407.095} C_VEL
LIN {X 0,Y 553.021,Z 299.123,A -85,B 0,C 180,E1 -3407.36,E2 -3407.36} C_VEL
LIN {X 0,Y 552.856,Z 310.861,A -85,B 0,C 180,E1 -3407.753,E2 -3407.753} C_VEL
LIN {X 0,Y 552.707,Z 320.382,A -85,B 0,C 180,E1 -3408.168,E2 -3408.168} C_VEL
LIN {X 0,Y 552.582,Z 330.488,A -85,B 0,C 180,E1 -3408.725,E2 -3408.725} C_VEL
LIN {X 0,Y 552.436,Z 340.022,A -85,B 0,C 180,E1 -3409.37,E2 -3409.37} C_VEL
LIN {X 0,Y 552.302,Z 348.001,A -85,B 0,C 180,E1 -3410.016,E2 -3410.016} C_VEL
LIN {X 0,Y 552.135,Z 356.601,A -85,B 0,C 180,E1 -3410.845,E2 -3410.845} C_VEL
LIN {X 0,Y 552.006,Z 364.54,A -85,B 0,C 180,E1 -3411.765,E2 -3411.765} C_VEL
LIN {X 0,Y 551.891,Z 372.474,A -85,B 0,C 180,E1 -3412.886,E2 -3412.886} C_VEL
LIN {X 0,Y 551.868,Z 379.419,A -85,B 0,C 180,E1 -3414.153,E2 -3414.153} C_VEL
LIN {X 0,Y 551.724,Z 384.147,A -85,B 0,C 180,E1 -3415.251,E2 -3415.251} C_VEL
LIN {X 0,Y 551.75,Z 387.779,A -85,B 0,C 180,E1 -3416.348,E2 -3416.348} C_VEL
LIN {X 0,Y 551.723,Z 389.672,A -85,B 0,C 180,E1 -3417.079,E2 -3417.079} C_VEL
LIN {X 0,Y 551.657,Z 391.135,A -85,B 0,C 180,E1 -3417.81,E2 -3417.81} C_VEL
LIN {X 0,Y 551.642,Z 392.732,A -85,B 0,C 180,E1 -3419.27,E2 -3419.27} C_VEL
LIN {X 0,Y 551.641,Z 392.996,A -85,B 0,C 180,E1 -3420,E2 -3420} C_VEL
LIN {X 0,Y 551.646,Z 392.205,A -85,B 0,C 180,E1 -3421.46,E2 -3421.46} C_VEL
LIN {X 0,Y 551.657,Z 391.281,A -85,B 0,C 180,E1 -3422.19,E2 -3422.19} C_VEL
LIN {X 0,Y 551.751,Z 388.035,A -85,B 0,C 180,E1 -3423.652,E2 -3423.652} C_VEL
LIN {X 0,Y 551.724,Z 384.485,A -85,B 0,C 180,E1 -3424.75,E2 -3424.75} C_VEL
LIN {X 0,Y 551.837,Z 379.838,A -85,B 0,C 180,E1 -3425.848,E2 -3425.848} C_VEL
LIN {X 0,Y 551.835,Z 375.027,A -85,B 0,C 180,E1 -3426.766,E2 -3426.766} C_VEL
LIN {X 0,Y 551.947,Z 369.233,A -85,B 0,C 180,E1 -3427.683,E2 -3427.683} C_VEL
LIN {X 0,Y 552.059,Z 362.28,A -85,B 0,C 180,E1 -3428.603,E2 -3428.603} C_VEL
LIN {X 0,Y 552.152,Z 355.693,A -85,B 0,C 180,E1 -3429.34,E2 -3429.34} C_VEL
LIN {X 0,Y 552.279,Z 347.966,A -85,B 0,C 180,E1 -3430.077,E2 -3430.077} C_VEL
LIN {X 0,Y 552.434,Z 339.982,A -85,B 0,C 180,E1 -3430.723,E2 -3430.723} C_VEL
LIN {X 0,Y 552.534,Z 331.948,A -85,B 0,C 180,E1 -3431.275,E2 -3431.275} C_VEL
LIN {X 0,Y 552.645,Z 323.967,A -85,B 0,C 180,E1 -3431.74,E2 -3431.74} C_VEL
LIN {X 0,Y 552.817,Z 313.068,A -85,B 0,C 180,E1 -3432.248,E2 -3432.248} C_VEL
LIN {X 0,Y 552.966,Z 302.73,A -85,B 0,C 180,E1 -3432.618,E2 -3432.618} C_VEL
LIN {X 0,Y 552.822,Z 296.845,A -85,B 0,C 180,E1 -3432.796,E2 -3432.796} C_VEL
LIN {X 0,Y 551.649,Z 289.891,A -85,B 0,C 180,E1 -3432.999,E2 -3432.999} C_VEL
LIN {X 0,Y 551.646,Z 286.995,A -85,B 0,C 180,E1 -3435.518,E2 -3435.518} C_VEL
LIN {X 0,Y 551.66,Z 284.554,A -85,B 0,C 180,E1 -3437.804,E2 -3437.804} C_VEL
LIN {X 0,Y 551.718,Z 282.275,A -85,B 0,C 180,E1 -3440.117,E2 -3440.117} C_VEL
LIN {X 0,Y 551.766,Z 280.759,A -85,B 0,C 180,E1 -3441.678,E2 -3441.678} C_VEL
LIN {X 0,Y 551.963,Z 280.732,A -85,B 0,C 180,E1 -3444.045,E2 -3444.045} C_VEL
LIN {X 0,Y 552.12,Z 280.709,A -85,B 0,C 180,E1 -3446.707,E2 -3446.707} C_VEL
LIN {X 0,Y 552.112,Z 280.71,A -85,B 0,C 180,E1 -3448.928,E2 -3448.928} C_VEL
LIN {X 0,Y 552.112,Z 280.708,A -85,B 0,C 180,E1 -3449.879,E2 -3449.879} C_VEL
LIN {X 0,Y 551.464,Z 280.795,A -85,B 0,C 180,E1 -3450.488,E2 -3450.488} C_VEL
LIN {X 0,Y 548.634,Z 281.147,A -85,B 0,C 180,E1 -3451.477,E2 -3451.477} C_VEL
LIN {X 0,Y 546.223,Z 281.446,A -85,B 0,C 180,E1 -3452.272,E2 -3452.272} C_VEL
LIN {X 0,Y 545.171,Z 281.575,A -85,B 0,C 180,E1 -3452.887,E2 -3452.887} C_VEL
LIN {X 0,Y 545.078,Z 281.584,A -85,B 0,C 180,E1 -3453.095,E2 -3453.095} C_VEL
LIN {X 0,Y 545.037,Z 281.588,A -85,B 0,C 180,E1 -3455.673,E2 -3455.673} C_VEL
LIN {X 0,Y 545.057,Z 281.594,A -85,B 0,C 180,E1 -3458.237,E2 -3458.237} C_VEL
LIN {X 0,Y 545.088,Z 281.583,A -85,B 0,C 180,E1 -3461.114,E2 -3461.114} C_VEL
LIN {X 0,Y 545.063,Z 281.591,A -85,B 0,C 180,E1 -3464.129,E2 -3464.129} C_VEL
LIN {X 0,Y 545.082,Z 281.582,A -85,B 0,C 180,E1 -3466.893,E2 -3466.893} C_VEL
LIN {X 0,Y 545.069,Z 281.592,A -85,B 0,C 180,E1 -3469.857,E2 -3469.857} C_VEL
LIN {X 0,Y 545.073,Z 281.586,A -85,B 0,C 180,E1 -3473.074,E2 -3473.074} C_VEL
LIN {X 0,Y 544.955,Z 281.608,A -85,B 0,C 180,E1 -3475.987,E2 -3475.987} C_VEL
LIN {X 0,Y 544.84,Z 287.123,A -85,B 0,C 180,E1 -3478.938,E2 -3478.938} C_VEL
LIN {X 0,Y 544.827,Z 291.604,A -85,B 0,C 180,E1 -3481.492,E2 -3481.492} C_VEL
LIN {X 0,Y 544.834,Z 296.904,A -85,B 0,C 180,E1 -3484.55,E2 -3484.55} C_VEL
LIN {X 0,Y 544.752,Z 301.634,A -85,B 0,C 180,E1 -3487.23,E2 -3487.23} C_VEL
LIN {X 0,Y 544.738,Z 307.259,A -85,B 0,C 180,E1 -3490.401,E2 -3490.401} C_VEL
LIN {X 0,Y 544.677,Z 312.663,A -85,B 0,C 180,E1 -3493.509,E2 -3493.509} C_VEL
LIN {X 0,Y 544.664,Z 316.715,A -85,B 0,C 180,E1 -3495.808,E2 -3495.808} C_VEL
LIN {X 0,Y 544.611,Z 318.657,A -85,B 0,C 180,E1 -3496.924,E2 -3496.924} C_VEL
LIN {X 0,Y 546.103,Z 327.996,A -85,B 0,C 180,E1 -3497.174,E2 -3497.174} C_VEL
LIN {X 0,Y 545.987,Z 337.063,A -85,B 0,C 180,E1 -3497.454,E2 -3497.454} C_VEL
LIN {X 0,Y 545.808,Z 347.398,A -85,B 0,C 180,E1 -3497.875,E2 -3497.875} C_VEL
LIN {X 0,Y 545.646,Z 356.28,A -85,B 0,C 180,E1 -3498.33,E2 -3498.33} C_VEL
LIN {X 0,Y 545.535,Z 364.802,A -85,B 0,C 180,E1 -3498.858,E2 -3498.858} C_VEL
LIN {X 0,Y 545.39,Z 373.61,A -85,B 0,C 180,E1 -3499.513,E2 -3499.513} C_VEL
LIN {X 0,Y 545.232,Z 381.064,A -85,B 0,C 180,E1 -3500.166,E2 -3500.166} C_VEL
LIN {X 0,Y 545.101,Z 388.326,A -85,B 0,C 180,E1 -3500.913,E2 -3500.913} C_VEL
LIN {X 0,Y 544.922,Z 395.932,A -85,B 0,C 180,E1 -3501.844,E2 -3501.844} C_VEL
LIN {X 0,Y 544.83,Z 402.274,A -85,B 0,C 180,E1 -3502.775,E2 -3502.775} C_VEL
LIN {X 0,Y 544.724,Z 407.354,A -85,B 0,C 180,E1 -3503.665,E2 -3503.665} C_VEL
LIN {X 0,Y 544.739,Z 411.153,A -85,B 0,C 180,E1 -3504.447,E2 -3504.447} C_VEL
LIN {X 0,Y 544.664,Z 415.487,A -85,B 0,C 180,E1 -3505.56,E2 -3505.56} C_VEL
LIN {X 0,Y 544.669,Z 417.851,A -85,B 0,C 180,E1 -3506.301,E2 -3506.301} C_VEL
LIN {X 0,Y 544.65,Z 419.657,A -85,B 0,C 180,E1 -3507.041,E2 -3507.041} C_VEL
LIN {X 0,Y 544.546,Z 422.15,A -85,B 0,C 180,E1 -3508.521,E2 -3508.521} C_VEL
LIN {X 0,Y 544.542,Z 422.741,A -85,B 0,C 180,E1 -3509.261,E2 -3509.261} C_VEL
LIN {X 0,Y 544.542,Z 422.808,A -85,B 0,C 180,E1 -3510.739,E2 -3510.739} C_VEL
LIN {X 0,Y 544.547,Z 422.228,A -85,B 0,C 180,E1 -3511.479,E2 -3511.479} C_VEL
LIN {X 0,Y 544.651,Z 419.874,A -85,B 0,C 180,E1 -3512.959,E2 -3512.959} C_VEL
LIN {X 0,Y 544.684,Z 416.988,A -85,B 0,C 180,E1 -3514.069,E2 -3514.069} C_VEL
LIN {X 0,Y 544.653,Z 413.071,A -85,B 0,C 180,E1 -3515.182,E2 -3515.182} C_VEL
LIN {X 0,Y 544.76,Z 408.872,A -85,B 0,C 180,E1 -3516.129,E2 -3516.129} C_VEL
LIN {X 0,Y 544.823,Z 402.829,A -85,B 0,C 180,E1 -3517.225,E2 -3517.225} C_VEL
LIN {X 0,Y 544.918,Z 396.593,A -85,B 0,C 180,E1 -3518.156,E2 -3518.156} C_VEL
LIN {X 0,Y 545.077,Z 389.106,A -85,B 0,C 180,E1 -3519.088,E2 -3519.088} C_VEL
LIN {X 0,Y 545.211,Z 381.983,A -85,B 0,C 180,E1 -3519.834,E2 -3519.834} C_VEL
LIN {X 0,Y 545.4,Z 373.563,A -85,B 0,C 180,E1 -3520.581,E2 -3520.581} C_VEL
LIN {X 0,Y 545.534,Z 364.289,A -85,B 0,C 180,E1 -3521.268,E2 -3521.268} C_VEL
LIN {X 0,Y 545.738,Z 352.29,A -85,B 0,C 180,E1 -3521.985,E2 -3521.985} C_VEL
LIN {X 0,Y 545.913,Z 340.801,A -85,B 0,C 180,E1 -3522.5,E2 -3522.5} C_VEL
LIN {X 0,Y 546.087,Z 329.575,A -85,B 0,C 180,E1 -3522.874,E2 -3522.874} C_VEL
LIN {X 0,Y 545.729,Z 324.985,A -85,B 0,C 180,E1 -3523.007,E2 -3523.007} C_VEL
LIN {X 0,Y 544.62,Z 318.618,A -85,B 0,C 180,E1 -3523.17,E2 -3523.17} C_VEL
LIN {X 0,Y 544.667,Z 314.174,A -85,B 0,C 180,E1 -3525.722,E2 -3525.722} C_VEL
LIN {X 0,Y 544.666,Z 310.175,A -85,B 0,C 180,E1 -3528.04,E2 -3528.04} C_VEL
LIN {X 0,Y 544.718,Z 306.039,A -85,B 0,C 180,E1 -3530.387,E2 -3530.387} C_VEL
LIN {X 0,Y 544.754,Z 301.811,A -85,B 0,C 180,E1 -3532.77,E2 -3532.77} C_VEL
LIN {X 0,Y 544.833,Z 297.063,A -85,B 0,C 180,E1 -3535.45,E2 -3535.45} C_VEL
LIN {X 0,Y 544.828,Z 291.762,A -85,B 0,C 180,E1 -3538.508,E2 -3538.508} C_VEL
LIN {X 0,Y 544.879,Z 286.214,A -85,B 0,C 180,E1 -3541.648,E2 -3541.648} C_VEL
LIN {X 0,Y 544.971,Z 281.605,A -85,B 0,C 180,E1 -3544.209,E2 -3544.209} C_VEL
LIN {X 0,Y 545.068,Z 281.591,A -85,B 0,C 180,E1 -3546.925,E2 -3546.925} C_VEL
LIN {X 0,Y 545.107,Z 281.585,A -85,B 0,C 180,E1 -3549.324,E2 -3549.324} C_VEL
LIN {X 0,Y 545.08,Z 281.589,A -85,B 0,C 180,E1 -3552.103,E2 -3552.103} C_VEL
LIN {X 0,Y 545.036,Z 281.596,A -85,B 0,C 180,E1 -3555.17,E2 -3555.17} C_VEL
LIN {X 0,Y 545.08,Z 281.589,A -85,B 0,C 180,E1 -3557.897,E2 -3557.897} C_VEL
LIN {X 0,Y 545.086,Z 281.587,A -85,B 0,C 180,E1 -3560.819,E2 -3560.819} C_VEL
LIN {X 0,Y 545.037,Z 281.594,A -85,B 0,C 180,E1 -3563.619,E2 -3563.619} C_VEL
LIN {X 0,Y 544.911,Z 281.684,A -85,B 0,C 180,E1 -3566.15,E2 -3566.15} C_VEL
LIN {X 0,Y 544.814,Z 286.81,A -85,B 0,C 180,E1 -3568.936,E2 -3568.936} C_VEL
LIN {X 0,Y 544.806,Z 291.415,A -85,B 0,C 180,E1 -3571.491,E2 -3571.491} C_VEL
LIN {X 0,Y 544.834,Z 296.921,A -85,B 0,C 180,E1 -3574.55,E2 -3574.55} C_VEL
LIN {X 0,Y 544.744,Z 301.653,A -85,B 0,C 180,E1 -3577.229,E2 -3577.229} C_VEL
LIN {X 0,Y 544.723,Z 305.841,A -85,B 0,C 180,E1 -3579.613,E2 -3579.613} C_VEL
LIN {X 0,Y 544.7,Z 311.428,A -85,B 0,C 180,E1 -3582.737,E2 -3582.737} C_VEL
LIN {X 0,Y 544.664,Z 316.666,A -85,B 0,C 180,E1 -3585.808,E2 -3585.808} C_VEL
LIN {X 0,Y 544.605,Z 318.689,A -85,B 0,C 180,E1 -3586.924,E2 -3586.924} C_VEL
LIN {X 0,Y 546.124,Z 328.065,A -85,B 0,C 180,E1 -3587.174,E2 -3587.174} C_VEL
LIN {X 0,Y 545.958,Z 341.051,A -85,B 0,C 180,E1 -3587.595,E2 -3587.595} C_VEL
LIN {X 0,Y 545.734,Z 352.228,A -85,B 0,C 180,E1 -3588.109,E2 -3588.109} C_VEL
LIN {X 0,Y 545.594,Z 360.82,A -85,B 0,C 180,E1 -3588.595,E2 -3588.595} C_VEL
LIN {X 0,Y 545.442,Z 370.067,A -85,B 0,C 180,E1 -3589.232,E2 -3589.232} C_VEL
LIN {X 0,Y 545.252,Z 379.054,A -85,B 0,C 180,E1 -3589.979,E2 -3589.979} C_VEL
LIN {X 0,Y 545.12,Z 386.62,A -85,B 0,C 180,E1 -3590.726,E2 -3590.726} C_VEL
LIN {X 0,Y 545.007,Z 393.1,A -85,B 0,C 180,E1 -3591.472,E2 -3591.472} C_VEL
LIN {X 0,Y 544.865,Z 399.904,A -85,B 0,C 180,E1 -3592.403,E2 -3592.403} C_VEL
LIN {X 0,Y 544.752,Z 406.029,A -85,B 0,C 180,E1 -3593.416,E2 -3593.416} C_VEL
LIN {X 0,Y 544.74,Z 411.117,A -85,B 0,C 180,E1 -3594.447,E2 -3594.447} C_VEL
LIN {X 0,Y 544.664,Z 415.469,A -85,B 0,C 180,E1 -3595.56,E2 -3595.56} C_VEL
LIN {X 0,Y 544.669,Z 417.831,A -85,B 0,C 180,E1 -3596.301,E2 -3596.301} C_VEL
LIN {X 0,Y 544.65,Z 419.686,A -85,B 0,C 180,E1 -3597.041,E2 -3597.041} C_VEL
LIN {X 0,Y 544.546,Z 422.129,A -85,B 0,C 180,E1 -3598.521,E2 -3598.521} C_VEL
LIN {X 0,Y 544.542,Z 422.761,A -85,B 0,C 180,E1 -3599.26,E2 -3599.26} C_VEL
LIN {X 0,Y 544.542,Z 422.794,A -85,B 0,C 180,E1 -3600.739,E2 -3600.739} C_VEL
LIN {X 0,Y 544.547,Z 422.24,A -85,B 0,C 180,E1 -3601.479,E2 -3601.479} C_VEL
LIN {X 0,Y 544.651,Z 419.867,A -85,B 0,C 180,E1 -3602.959,E2 -3602.959} C_VEL
LIN {X 0,Y 544.684,Z 416.986,A -85,B 0,C 180,E1 -3604.069,E2 -3604.069} C_VEL
LIN {X 0,Y 544.653,Z 413.071,A -85,B 0,C 180,E1 -3605.182,E2 -3605.182} C_VEL
LIN {X 0,Y 544.762,Z 408.875,A -85,B 0,C 180,E1 -3606.129,E2 -3606.129} C_VEL
LIN {X 0,Y 544.822,Z 402.832,A -85,B 0,C 180,E1 -3607.225,E2 -3607.225} C_VEL
LIN {X 0,Y 544.915,Z 396.596,A -85,B 0,C 180,E1 -3608.156,E2 -3608.156} C_VEL
LIN {X 0,Y 545.027,Z 390.744,A -85,B 0,C 180,E1 -3608.902,E2 -3608.902} C_VEL
LIN {X 0,Y 545.16,Z 383.926,A -85,B 0,C 180,E1 -3609.648,E2 -3609.648} C_VEL
LIN {X 0,Y 545.376,Z 374.705,A -85,B 0,C 180,E1 -3610.488,E2 -3610.488} C_VEL
LIN {X 0,Y 545.478,Z 366.106,A -85,B 0,C 180,E1 -3611.143,E2 -3611.143} C_VEL
LIN {X 0,Y 545.633,Z 356.942,A -85,B 0,C 180,E1 -3611.723,E2 -3611.723} C_VEL
LIN {X 0,Y 545.815,Z 347.335,A -85,B 0,C 180,E1 -3612.219,E2 -3612.219} C_VEL
LIN {X 0,Y 546.009,Z 336.948,A -85,B 0,C 180,E1 -3612.64,E2 -3612.64} C_VEL
LIN {X 0,Y 545.993,Z 326.518,A -85,B 0,C 180,E1 -3612.959,E2 -3612.959} C_VEL
LIN {X 0,Y 544.62,Z 318.624,A -85,B 0,C 180,E1 -3613.17,E2 -3613.17} C_VEL
LIN {X 0,Y 544.686,Z 314.326,A -85,B 0,C 180,E1 -3615.721,E2 -3615.721} C_VEL
LIN {X 0,Y 544.672,Z 310.302,A -85,B 0,C 180,E1 -3618.04,E2 -3618.04} C_VEL
LIN {X 0,Y 544.736,Z 306.119,A -85,B 0,C 180,E1 -3620.386,E2 -3620.386} C_VEL
LIN {X 0,Y 544.758,Z 301.813,A -85,B 0,C 180,E1 -3622.77,E2 -3622.77} C_VEL
LIN {X 0,Y 544.793,Z 296.678,A -85,B 0,C 180,E1 -3625.441,E2 -3625.441} C_VEL
LIN {X 0,Y 544.73,Z 292.167,A -85,B 0,C 180,E1 -3627.676,E2 -3627.676} C_VEL
LIN {X 0,Y 544.637,Z 286.549,A -85,B 0,C 180,E1 -3630.216,E2 -3630.216} C_VEL
LIN {X 0,Y 544.67,Z 281.643,A -85,B 0,C 180,E1 -3632.267,E2 -3632.267} C_VEL
LIN {X 0,Y 545.035,Z 281.595,A -85,B 0,C 180,E1 -3634.385,E2 -3634.385} C_VEL
LIN {X 0,Y 545.037,Z 281.594,A -85,B 0,C 180,E1 -3637.304,E2 -3637.304} C_VEL
LIN {X 0,Y 545.067,Z 281.591,A -85,B 0,C 180,E1 -3640.143,E2 -3640.143} C_VEL
LIN {X 0,Y 545.05,Z 281.593,A -85,B 0,C 180,E1 -3642.695,E2 -3642.695} C_VEL
LIN {X 0,Y 545.065,Z 281.59,A -85,B 0,C 180,E1 -3645.167,E2 -3645.167} C_VEL
LIN {X 0,Y 545.078,Z 281.591,A -85,B 0,C 180,E1 -3648.403,E2 -3648.403} C_VEL
LIN {X 0,Y 545.081,Z 281.592,A -85,B 0,C 180,E1 -3650.818,E2 -3650.818} C_VEL
LIN {X 0,Y 545.054,Z 281.596,A -85,B 0,C 180,E1 -3651.864,E2 -3651.864} C_VEL
LIN {X 0,Y 546.423,Z 288.93,A -85,B 0,C 180,E1 -3654.125,E2 -3654.125} C_VEL
LIN {X 0,Y 546.248,Z 298.157,A -85,B 0,C 180,E1 -3656.75,E2 -3656.75} C_VEL
LIN {X 0,Y 546.002,Z 308.289,A -85,B 0,C 180,E1 -3659.588,E2 -3659.588} C_VEL
LIN {X 0,Y 545.769,Z 318.502,A -85,B 0,C 180,E1 -3662.381,E2 -3662.381} C_VEL
LIN {X 0,Y 545.568,Z 327.71,A -85,B 0,C 180,E1 -3664.843,E2 -3664.843} C_VEL
LIN {X 0,Y 545.42,Z 336.919,A -85,B 0,C 180,E1 -3667.259,E2 -3667.259} C_VEL
LIN {X 0,Y 545.244,Z 349.197,A -85,B 0,C 180,E1 -3670.419,E2 -3670.419} C_VEL
LIN {X 0,Y 545.078,Z 359.94,A -85,B 0,C 180,E1 -3673.136,E2 -3673.136} C_VEL
LIN {X 0,Y 544.922,Z 372.218,A -85,B 0,C 180,E1 -3676.196,E2 -3676.196} C_VEL
LIN {X 0,Y 544.879,Z 374.712,A -85,B 0,C 180,E1 -3676.812,E2 -3676.812} C_VEL
LIN {X 0,Y 546.193,Z 383.507,A -85,B 0,C 180,E1 -3677.01,E2 -3677.01} C_VEL
LIN {X 0,Y 546.018,Z 395.875,A -85,B 0,C 180,E1 -3677.361,E2 -3677.361} C_VEL
LIN {X 0,Y 545.827,Z 407.508,A -85,B 0,C 180,E1 -3677.828,E2 -3677.828} C_VEL
LIN {X 0,Y 545.62,Z 419.862,A -85,B 0,C 180,E1 -3678.488,E2 -3678.488} C_VEL
LIN {X 0,Y 545.422,Z 430.746,A -85,B 0,C 180,E1 -3679.232,E2 -3679.232} C_VEL
LIN {X 0,Y 545.227,Z 441.601,A -85,B 0,C 180,E1 -3680.166,E2 -3680.166} C_VEL
LIN {X 0,Y 545.051,Z 450.412,A -85,B 0,C 180,E1 -3681.099,E2 -3681.099} C_VEL
LIN {X 0,Y 544.896,Z 459.001,A -85,B 0,C 180,E1 -3682.217,E2 -3682.217} C_VEL
LIN {X 0,Y 544.745,Z 466.35,A -85,B 0,C 180,E1 -3683.421,E2 -3683.421} C_VEL
LIN {X 0,Y 544.741,Z 471.366,A -85,B 0,C 180,E1 -3684.447,E2 -3684.447} C_VEL
LIN {X 0,Y 544.66,Z 475.677,A -85,B 0,C 180,E1 -3685.56,E2 -3685.56} C_VEL
LIN {X 0,Y 544.669,Z 477.957,A -85,B 0,C 180,E1 -3686.301,E2 -3686.301} C_VEL
LIN {X 0,Y 544.65,Z 479.808,A -85,B 0,C 180,E1 -3687.041,E2 -3687.041} C_VEL
LIN {X 0,Y 544.546,Z 482.185,A -85,B 0,C 180,E1 -3688.521,E2 -3688.521} C_VEL
LIN {X 0,Y 544.541,Z 483,A -85,B 0,C 180,E1 -3690,E2 -3690} C_VEL
LIN {X 0,Y 544.546,Z 482.186,A -85,B 0,C 180,E1 -3691.479,E2 -3691.479} C_VEL
LIN {X 0,Y 544.65,Z 479.81,A -85,B 0,C 180,E1 -3692.959,E2 -3692.959} C_VEL
LIN {X 0,Y 544.684,Z 476.896,A -85,B 0,C 180,E1 -3694.069,E2 -3694.069} C_VEL
LIN {X 0,Y 544.653,Z 472.949,A -85,B 0,C 180,E1 -3695.182,E2 -3695.182} C_VEL
LIN {X 0,Y 544.737,Z 467.595,A -85,B 0,C 180,E1 -3696.349,E2 -3696.349} C_VEL
LIN {X 0,Y 544.859,Z 460.237,A -85,B 0,C 180,E1 -3697.597,E2 -3697.597} C_VEL
LIN {X 0,Y 545.029,Z 451.99,A -85,B 0,C 180,E1 -3698.715,E2 -3698.715} C_VEL
LIN {X 0,Y 545.164,Z 443.538,A -85,B 0,C 180,E1 -3699.648,E2 -3699.648} C_VEL
LIN {X 0,Y 545.419,Z 433.097,A -85,B 0,C 180,E1 -3700.581,E2 -3700.581} C_VEL
LIN {X 0,Y 545.605,Z 421.663,A -85,B 0,C 180,E1 -3701.401,E2 -3701.401} C_VEL
LIN {X 0,Y 545.761,Z 411.41,A -85,B 0,C 180,E1 -3701.985,E2 -3701.985} C_VEL
LIN {X 0,Y 545.941,Z 399.762,A -85,B 0,C 180,E1 -3702.5,E2 -3702.5} C_VEL
LIN {X 0,Y 546.122,Z 386.346,A -85,B 0,C 180,E1 -3702.92,E2 -3702.92} C_VEL
LIN {X 0,Y 545.973,Z 381.512,A -85,B 0,C 180,E1 -3703.036,E2 -3703.036} C_VEL
LIN {X 0,Y 544.879,Z 374.712,A -85,B 0,C 180,E1 -3703.188,E2 -3703.188} C_VEL
LIN {X 0,Y 544.996,Z 363.009,A -85,B 0,C 180,E1 -3706.096,E2 -3706.096} C_VEL
LIN {X 0,Y 545.191,Z 352.266,A -85,B 0,C 180,E1 -3708.801,E2 -3708.801} C_VEL
LIN {X 0,Y 545.38,Z 339.988,A -85,B 0,C 180,E1 -3711.945,E2 -3711.945} C_VEL
LIN {X 0,Y 545.525,Z 330.78,A -85,B 0,C 180,E1 -3714.347,E2 -3714.347} C_VEL
LIN {X 0,Y 545.704,Z 321.571,A -85,B 0,C 180,E1 -3716.792,E2 -3716.792} C_VEL
LIN {X 0,Y 545.964,Z 310.828,A -85,B 0,C 180,E1 -3719.709,E2 -3719.709} C_VEL
LIN {X 0,Y 546.183,Z 301.621,A -85,B 0,C 180,E1 -3722.276,E2 -3722.276} C_VEL
LIN {X 0,Y 546.305,Z 291.831,A -85,B 0,C 180,E1 -3724.932,E2 -3724.932} C_VEL
LIN {X 0,Y 546.046,Z 286.884,A -85,B 0,C 180,E1 -3726.303,E2 -3726.303} C_VEL
LIN {X 0,Y 545.072,Z 281.591,A -85,B 0,C 180,E1 -3727.943,E2 -3727.943} C_VEL
LIN {X 0,Y 545.08,Z 281.591,A -85,B 0,C 180,E1 -3730.472,E2 -3730.472} C_VEL
LIN {X 0,Y 545.024,Z 281.596,A -85,B 0,C 180,E1 -3733.112,E2 -3733.112} C_VEL
LIN {X 0,Y 545.051,Z 281.594,A -85,B 0,C 180,E1 -3736.226,E2 -3736.226} C_VEL
LIN {X 0,Y 545.082,Z 281.587,A -85,B 0,C 180,E1 -3738.885,E2 -3738.885} C_VEL
LIN {X 0,Y 545.086,Z 281.586,A -85,B 0,C 180,E1 -3740.819,E2 -3740.819} C_VEL
LIN {X 0,Y 545.045,Z 281.592,A -85,B 0,C 180,E1 -3743.62,E2 -3743.62} C_VEL
LIN {X 0,Y 545.069,Z 281.589,A -85,B 0,C 180,E1 -3746.328,E2 -3746.328} C_VEL
LIN {X 0,Y 545.069,Z 281.587,A -85,B 0,C 180,E1 -3748.952,E2 -3748.952} C_VEL
LIN {X 0,Y 545.105,Z 281.589,A -85,B 0,C 180,E1 -3751.508,E2 -3751.508} C_VEL
LIN {X 0,Y 545.071,Z 281.589,A -85,B 0,C 180,E1 -3753.999,E2 -3753.999} C_VEL
LIN {X 0,Y 544.962,Z 281.607,A -85,B 0,C 180,E1 -3756.435,E2 -3756.435} C_VEL
LIN {X 0,Y 544.84,Z 281.622,A -85,B 0,C 180,E1 -3757.233,E2 -3757.233} C_VEL
LIN {X 0,Y 544.804,Z 283.763,A -85,B 0,C 180,E1 -3759.617,E2 -3759.617} C_VEL
LIN {X 0,Y 544.7,Z 286.469,A -85,B 0,C 180,E1 -3762.737,E2 -3762.737} C_VEL
LIN {X 0,Y 544.643,Z 289.209,A -85,B 0,C 180,E1 -3765.808,E2 -3765.808} C_VEL
LIN {X 0,Y 544.59,Z 290.284,A -85,B 0,C 180,E1 -3766.948,E2 -3766.948} C_VEL
LIN {X 0,Y 546.092,Z 299.879,A -85,B 0,C 180,E1 -3767.221,E2 -3767.221} C_VEL
LIN {X 0,Y 545.903,Z 310.856,A -85,B 0,C 180,E1 -3767.594,E2 -3767.594} C_VEL
LIN {X 0,Y 545.767,Z 320.374,A -85,B 0,C 180,E1 -3768.016,E2 -3768.016} C_VEL
LIN {X 0,Y 545.587,Z 330.805,A -85,B 0,C 180,E1 -3768.599,E2 -3768.599} C_VEL
LIN {X 0,Y 545.427,Z 340.016,A -85,B 0,C 180,E1 -3769.232,E2 -3769.232} C_VEL
LIN {X 0,Y 545.261,Z 347.996,A -85,B 0,C 180,E1 -3769.886,E2 -3769.886} C_VEL
LIN {X 0,Y 545.157,Z 354.837,A -85,B 0,C 180,E1 -3770.539,E2 -3770.539} C_VEL
LIN {X 0,Y 545.019,Z 361.556,A -85,B 0,C 180,E1 -3771.285,E2 -3771.285} C_VEL
LIN {X 0,Y 544.896,Z 368.616,A -85,B 0,C 180,E1 -3772.217,E2 -3772.217} C_VEL
LIN {X 0,Y 544.796,Z 374.509,A -85,B 0,C 180,E1 -3773.147,E2 -3773.147} C_VEL
LIN {X 0,Y 544.778,Z 379.413,A -85,B 0,C 180,E1 -3774.076,E2 -3774.076} C_VEL
LIN {X 0,Y 544.628,Z 384.141,A -85,B 0,C 180,E1 -3775.189,E2 -3775.189} C_VEL
LIN {X 0,Y 544.669,Z 387.774,A -85,B 0,C 180,E1 -3776.301,E2 -3776.301} C_VEL
LIN {X 0,Y 544.65,Z 389.667,A -85,B 0,C 180,E1 -3777.041,E2 -3777.041} C_VEL
LIN {X 0,Y 544.572,Z 391.134,A -85,B 0,C 180,E1 -3777.781,E2 -3777.781} C_VEL
LIN {X 0,Y 544.542,Z 392.725,A -85,B 0,C 180,E1 -3779.261,E2 -3779.261} C_VEL
LIN {X 0,Y 544.542,Z 392.996,A -85,B 0,C 180,E1 -3780,E2 -3780} C_VEL
LIN {X 0,Y 544.547,Z 392.196,A -85,B 0,C 180,E1 -3781.479,E2 -3781.479} C_VEL
LIN {X 0,Y 544.572,Z 391.281,A -85,B 0,C 180,E1 -3782.219,E2 -3782.219} C_VEL
LIN {X 0,Y 544.669,Z 388.027,A -85,B 0,C 180,E1 -3783.699,E2 -3783.699} C_VEL
LIN {X 0,Y 544.628,Z 384.475,A -85,B 0,C 180,E1 -3784.812,E2 -3784.812} C_VEL
LIN {X 0,Y 544.754,Z 379.827,A -85,B 0,C 180,E1 -3785.924,E2 -3785.924} C_VEL
LIN {X 0,Y 544.762,Z 375.014,A -85,B 0,C 180,E1 -3786.854,E2 -3786.854} C_VEL
LIN {X 0,Y 544.872,Z 369.22,A -85,B 0,C 180,E1 -3787.784,E2 -3787.784} C_VEL
LIN {X 0,Y 544.994,Z 362.266,A -85,B 0,C 180,E1 -3788.715,E2 -3788.715} C_VEL
LIN {X 0,Y 545.13,Z 355.678,A -85,B 0,C 180,E1 -3789.461,E2 -3789.461} C_VEL
LIN {X 0,Y 545.277,Z 347.948,A -85,B 0,C 180,E1 -3790.208,E2 -3790.208} C_VEL
LIN {X 0,Y 545.444,Z 339.96,A -85,B 0,C 180,E1 -3790.862,E2 -3790.862} C_VEL
LIN {X 0,Y 545.583,Z 330.769,A -85,B 0,C 180,E1 -3791.493,E2 -3791.493} C_VEL
LIN {X 0,Y 545.758,Z 322.095,A -85,B 0,C 180,E1 -3791.985,E2 -3791.985} C_VEL
LIN {X 0,Y 545.886,Z 313.03,A -85,B 0,C 180,E1 -3792.406,E2 -3792.406} C_VEL
LIN {X 0,Y 546.021,Z 303.459,A -85,B 0,C 180,E1 -3792.757,E2 -3792.757} C_VEL
LIN {X 0,Y 545.862,Z 297.281,A -85,B 0,C 180,E1 -3792.95,E2 -3792.95} C_VEL
LIN {X 0,Y 544.568,Z 290.059,A -85,B 0,C 180,E1 -3793.148,E2 -3793.148} C_VEL
LIN {X 0,Y 544.574,Z 287.404,A -85,B 0,C 180,E1 -3795.725,E2 -3795.725} C_VEL
LIN {X 0,Y 544.59,Z 285.068,A -85,B 0,C 180,E1 -3798.043,E2 -3798.043} C_VEL
LIN {X 0,Y 544.637,Z 282.541,A -85,B 0,C 180,E1 -3800.39,E2 -3800.39} C_VEL
LIN {X 0,Y 544.647,Z 281.705,A -85,B 0,C 180,E1 -3801.181,E2 -3801.181} C_VEL
LIN {X 0,Y 544.909,Z 281.613,A -85,B 0,C 180,E1 -3803.69,E2 -3803.69} C_VEL
LIN {X 0,Y 545.069,Z 281.584,A -85,B 0,C 180,E1 -3806.001,E2 -3806.001} C_VEL
LIN {X 0,Y 545.092,Z 281.587,A -85,B 0,C 180,E1 -3808.748,E2 -3808.748} C_VEL
